LIN {X 0,Y 125.306,Z 694.835,A -85,B 0,C 180,E1 -25457.036,E2 -25457.036} C_VEL
LIN {X 0,Y 123.812,Z 697.112,A -85,B 0,C 180,E1 -25463.481,E2 -25463.481} C_VEL
LIN {X 0,Y 123.139,Z 697.936,A -85,B 0,C 180,E1 -25470,E2 -25470} C_VEL
LIN {X 0,Y 123.809,Z 697.16,A -85,B 0,C 180,E1 -25476.519,E2 -25476.519} C_VEL
LIN {X 0,Y 125.288,Z 694.933,A -85,B 0,C 180,E1 -25482.966,E2 -25482.966} C_VEL
LIN {X 0,Y 127.632,Z 692.097,A -85,B 0,C 180,E1 -25487.629,E2 -25487.629} C_VEL
LIN {X 0,Y 130.588,Z 688.261,A -85,B 0,C 180,E1 -25492.13,E2 -25492.13} C_VEL
LIN {X 0,Y 134.038,Z 683.171,A -85,B 0,C 180,E1 -25496.633,E2 -25496.633} C_VEL
LIN {X 0,Y 137.979,Z 677.127,A -85,B 0,C 180,E1 -25500.62,E2 -25500.62} C_VEL
LIN {X 0,Y 142.589,Z 669.335,A -85,B 0,C 180,E1 -25504.528,E2 -25504.528} C_VEL
LIN {X 0,Y 147.556,Z 659.65,A -85,B 0,C 180,E1 -25508.255,E2 -25508.255} C_VEL
LIN {X 0,Y 151.618,Z 650.591,A -85,B 0,C 180,E1 -25510.899,E2 -25510.899} C_VEL
LIN {X 0,Y 156.205,Z 639.02,A -85,B 0,C 180,E1 -25513.402,E2 -25513.402} C_VEL
LIN {X 0,Y 159.797,Z 627.372,A -85,B 0,C 180,E1 -25515.368,E2 -25515.368} C_VEL
LIN {X 0,Y 162.681,Z 615.545,A -85,B 0,C 180,E1 -25516.802,E2 -25516.802} C_VEL
LIN {X 0,Y 164.589,Z 602.681,A -85,B 0,C 180,E1 -25518.039,E2 -25518.039} C_VEL
LIN {X 0,Y 165.697,Z 590.213,A -85,B 0,C 180,E1 -25518.804,E2 -25518.804} C_VEL
LIN {X 0,Y 166.609,Z 571.79,A -85,B 0,C 180,E1 -25519.65,E2 -25519.65} C_VEL
LIN {X 0,Y 161.362,Z 561.441,A -85,B 0,C 180,E1 -25522.733,E2 -25522.733} C_VEL
LIN {X 0,Y 156.028,Z 552.146,A -85,B 0,C 180,E1 -25526.256,E2 -25526.256} C_VEL
LIN {X 0,Y 151.661,Z 545.284,A -85,B 0,C 180,E1 -25529.556,E2 -25529.556} C_VEL
LIN {X 0,Y 148.447,Z 540.617,A -85,B 0,C 180,E1 -25532.318,E2 -25532.318} C_VEL
LIN {X 0,Y 145.829,Z 537.015,A -85,B 0,C 180,E1 -25534.861,E2 -25534.861} C_VEL
LIN {X 0,Y 143.17,Z 533.482,A -85,B 0,C 180,E1 -25537.829,E2 -25537.829} C_VEL
LIN {X 0,Y 142.512,Z 532.415,A -85,B 0,C 180,E1 -25538.672,E2 -25538.672} C_VEL
LIN {X 0,Y 140.116,Z 529.937,A -85,B 0,C 180,E1 -25541.919,E2 -25541.919} C_VEL
LIN {X 0,Y 138.65,Z 527.238,A -85,B 0,C 180,E1 -25544.549,E2 -25544.549} C_VEL
LIN {X 0,Y 135.862,Z 524.714,A -85,B 0,C 180,E1 -25551.072,E2 -25551.072} C_VEL
LIN {X 0,Y 134.903,Z 522.132,A -85,B 0,C 180,E1 -25557.761,E2 -25557.761} C_VEL
LIN {X 0,Y 134.928,Z 521.81,A -85,B 0,C 180,E1 -25560,E2 -25560} C_VEL
LIN {X 0,Y 135.097,Z 522.892,A -85,B 0,C 180,E1 -25562.982,E2 -25562.982} C_VEL
LIN {X 0,Y 138.648,Z 527.444,A -85,B 0,C 180,E1 -25573.558,E2 -25573.558} C_VEL
LIN {X 0,Y 140.387,Z 530.729,A -85,B 0,C 180,E1 -25576.636,E2 -25576.636} C_VEL
LIN {X 0,Y 144.122,Z 537.229,A -85,B 0,C 180,E1 -25581.674,E2 -25581.674} C_VEL
LIN {X 0,Y 147.623,Z 543.935,A -85,B 0,C 180,E1 -25585.465,E2 -25585.465} C_VEL
LIN {X 0,Y 150.822,Z 550.425,A -85,B 0,C 180,E1 -25588.436,E2 -25588.436} C_VEL
LIN {X 0,Y 153.946,Z 557.142,A -85,B 0,C 180,E1 -25591.021,E2 -25591.021} C_VEL
LIN {X 0,Y 158.018,Z 566.743,A -85,B 0,C 180,E1 -25594.064,E2 -25594.064} C_VEL
LIN {X 0,Y 161.409,Z 576.189,A -85,B 0,C 180,E1 -25596.43,E2 -25596.43} C_VEL
LIN {X 0,Y 162.087,Z 578.257,A -85,B 0,C 180,E1 -25596.888,E2 -25596.888} C_VEL
LIN {X 0,Y 162.907,Z 608.203,A -85,B 0,C 180,E1 -25599.302,E2 -25599.302} C_VEL
LIN {X 0,Y 162.981,Z 619.724,A -85,B 0,C 180,E1 -25600.096,E2 -25600.096} C_VEL
LIN {X 0,Y 161.369,Z 633.381,A -85,B 0,C 180,E1 -25600.774,E2 -25600.774} C_VEL
LIN {X 0,Y 158.919,Z 645.815,A -85,B 0,C 180,E1 -25601.733,E2 -25601.733} C_VEL
LIN {X 0,Y 156.037,Z 656.834,A -85,B 0,C 180,E1 -25602.955,E2 -25602.955} C_VEL
LIN {X 0,Y 151.954,Z 668.683,A -85,B 0,C 180,E1 -25604.677,E2 -25604.677} C_VEL
LIN {X 0,Y 146.967,Z 680.536,A -85,B 0,C 180,E1 -25607.045,E2 -25607.045} C_VEL
LIN {X 0,Y 142.734,Z 689.116,A -85,B 0,C 180,E1 -25609.278,E2 -25609.278} C_VEL
LIN {X 0,Y 137.87,Z 698.049,A -85,B 0,C 180,E1 -25612.288,E2 -25612.288} C_VEL
LIN {X 0,Y 132.801,Z 706.821,A -85,B 0,C 180,E1 -25616.244,E2 -25616.244} C_VEL
LIN {X 0,Y 128.555,Z 713.893,A -85,B 0,C 180,E1 -25620.527,E2 -25620.527} C_VEL
LIN {X 0,Y 125.022,Z 719.59,A -85,B 0,C 180,E1 -25625.065,E2 -25625.065} C_VEL
LIN {X 0,Y 122.616,Z 724.144,A -85,B 0,C 180,E1 -25629.886,E2 -25629.886} C_VEL
LIN {X 0,Y 121.177,Z 727.643,A -85,B 0,C 180,E1 -25634.872,E2 -25634.872} C_VEL
LIN {X 0,Y 120.787,Z 730.791,A -85,B 0,C 180,E1 -25641.55,E2 -25641.55} C_VEL
LIN {X 0,Y 121.419,Z 732.086,A -85,B 0,C 180,E1 -25646.682,E2 -25646.682} C_VEL
LIN {X 0,Y 122.117,Z 732.42,A -85,B 0,C 180,E1 -25650,E2 -25650} C_VEL
LIN {X 0,Y 121.429,Z 732.072,A -85,B 0,C 180,E1 -25653.318,E2 -25653.318} C_VEL
LIN {X 0,Y 120.759,Z 730.143,A -85,B 0,C 180,E1 -25660.055,E2 -25660.055} C_VEL
LIN {X 0,Y 121.18,Z 727.586,A -85,B 0,C 180,E1 -25665.128,E2 -25665.128} C_VEL
LIN {X 0,Y 122.647,Z 724.065,A -85,B 0,C 180,E1 -25670.109,E2 -25670.109} C_VEL
LIN {X 0,Y 125.085,Z 719.488,A -85,B 0,C 180,E1 -25674.922,E2 -25674.922} C_VEL
LIN {X 0,Y 128.554,Z 713.754,A -85,B 0,C 180,E1 -25679.473,E2 -25679.473} C_VEL
LIN {X 0,Y 132.799,Z 706.649,A -85,B 0,C 180,E1 -25683.757,E2 -25683.757} C_VEL
LIN {X 0,Y 135.921,Z 701.383,A -85,B 0,C 180,E1 -25686.236,E2 -25686.236} C_VEL
LIN {X 0,Y 137.564,Z 697.485,A -85,B 0,C 180,E1 -25687.963,E2 -25687.963} C_VEL
LIN {X 0,Y 138.814,Z 690.741,A -85,B 0,C 180,E1 -25690.95,E2 -25690.95} C_VEL
LIN {X 0,Y 140.224,Z 683.56,A -85,B 0,C 180,E1 -25693.685,E2 -25693.685} C_VEL
LIN {X 0,Y 142.028,Z 678.907,A -85,B 0,C 180,E1 -25694.966,E2 -25694.966} C_VEL
LIN {X 0,Y 147.013,Z 667.262,A -85,B 0,C 180,E1 -25697.306,E2 -25697.306} C_VEL
LIN {X 0,Y 151.212,Z 655.339,A -85,B 0,C 180,E1 -25699.023,E2 -25699.023} C_VEL
LIN {X 0,Y 154.607,Z 642.61,A -85,B 0,C 180,E1 -25700.371,E2 -25700.371} C_VEL
LIN {X 0,Y 157.066,Z 629.589,A -85,B 0,C 180,E1 -25701.309,E2 -25701.309} C_VEL
LIN {X 0,Y 158.216,Z 618.69,A -85,B 0,C 180,E1 -25701.849,E2 -25701.849} C_VEL
LIN {X 0,Y 157.786,Z 586.961,A -85,B 0,C 180,E1 -25704.348,E2 -25704.348} C_VEL
LIN {X 0,Y 157.453,Z 580.228,A -85,B 0,C 180,E1 -25705.02,E2 -25705.02} C_VEL
LIN {X 0,Y 153.782,Z 569.769,A -85,B 0,C 180,E1 -25707.812,E2 -25707.812} C_VEL
LIN {X 0,Y 150.559,Z 561.823,A -85,B 0,C 180,E1 -25710.459,E2 -25710.459} C_VEL
LIN {X 0,Y 147.233,Z 554.175,A -85,B 0,C 180,E1 -25713.509,E2 -25713.509} C_VEL
LIN {X 0,Y 144.191,Z 547.823,A -85,B 0,C 180,E1 -25716.671,E2 -25716.671} C_VEL
LIN {X 0,Y 141.243,Z 541.932,A -85,B 0,C 180,E1 -25720.28,E2 -25720.28} C_VEL
LIN {X 0,Y 137.569,Z 534.878,A -85,B 0,C 180,E1 -25726.144,E2 -25726.144} C_VEL
LIN {X 0,Y 136.741,Z 533.764,A -85,B 0,C 180,E1 -25727.76,E2 -25727.76} C_VEL
LIN {X 0,Y 133.829,Z 528.876,A -85,B 0,C 180,E1 -25738.496,E2 -25738.496} C_VEL
LIN {X 0,Y 133.756,Z 528.586,A -85,B 0,C 180,E1 -25740,E2 -25740} C_VEL
LIN {X 0,Y 133.924,Z 529.552,A -85,B 0,C 180,E1 -25744.892,E2 -25744.892} C_VEL
LIN {X 0,Y 136.671,Z 533.761,A -85,B 0,C 180,E1 -25754.138,E2 -25754.138} C_VEL
LIN {X 0,Y 137.444,Z 534.332,A -85,B 0,C 180,E1 -25755.572,E2 -25755.572} C_VEL
LIN {X 0,Y 139.633,Z 537.994,A -85,B 0,C 180,E1 -25759.301,E2 -25759.301} C_VEL
LIN {X 0,Y 141.113,Z 539.535,A -85,B 0,C 180,E1 -25761.262,E2 -25761.262} C_VEL
LIN {X 0,Y 143.561,Z 543.129,A -85,B 0,C 180,E1 -25764.214,E2 -25764.214} C_VEL
LIN {X 0,Y 144.875,Z 544.981,A -85,B 0,C 180,E1 -25765.615,E2 -25765.615} C_VEL
LIN {X 0,Y 147.5,Z 548.879,A -85,B 0,C 180,E1 -25768.165,E2 -25768.165} C_VEL
LIN {X 0,Y 151.608,Z 555.279,A -85,B 0,C 180,E1 -25771.64,E2 -25771.64} C_VEL
LIN {X 0,Y 156.801,Z 564.449,A -85,B 0,C 180,E1 -25775.442,E2 -25775.442} C_VEL
LIN {X 0,Y 160.843,Z 572.43,A -85,B 0,C 180,E1 -25778.073,E2 -25778.073} C_VEL
LIN {X 0,Y 161.898,Z 574.617,A -85,B 0,C 180,E1 -25778.72,E2 -25778.72} C_VEL
LIN {X 0,Y 160.405,Z 598.06,A -85,B 0,C 180,E1 -25779.851,E2 -25779.851} C_VEL
LIN {X 0,Y 158.623,Z 611.11,A -85,B 0,C 180,E1 -25780.869,E2 -25780.869} C_VEL
LIN {X 0,Y 156.036,Z 623.487,A -85,B 0,C 180,E1 -25782.265,E2 -25782.265} C_VEL
LIN {X 0,Y 152.82,Z 634.629,A -85,B 0,C 180,E1 -25783.94,E2 -25783.94} C_VEL
LIN {X 0,Y 148.976,Z 644.988,A -85,B 0,C 180,E1 -25785.907,E2 -25785.907} C_VEL
LIN {X 0,Y 144.507,Z 655.294,A -85,B 0,C 180,E1 -25788.5,E2 -25788.5} C_VEL
LIN {X 0,Y 140.323,Z 663.695,A -85,B 0,C 180,E1 -25791.241,E2 -25791.241} C_VEL
LIN {X 0,Y 136.036,Z 671.414,A -85,B 0,C 180,E1 -25794.465,E2 -25794.465} C_VEL
LIN {X 0,Y 131.173,Z 679.072,A -85,B 0,C 180,E1 -25798.598,E2 -25798.598} C_VEL
LIN {X 0,Y 126.465,Z 685.867,A -85,B 0,C 180,E1 -25803.604,E2 -25803.604} C_VEL
LIN {X 0,Y 122.952,Z 690.47,A -85,B 0,C 180,E1 -25808.19,E2 -25808.19} C_VEL
LIN {X 0,Y 119.998,Z 694.005,A -85,B 0,C 180,E1 -25812.972,E2 -25812.972} C_VEL
LIN {X 0,Y 118.466,Z 695.825,A -85,B 0,C 180,E1 -25816.273,E2 -25816.273} C_VEL
LIN {X 0,Y 116.832,Z 698.101,A -85,B 0,C 180,E1 -25823.09,E2 -25823.09} C_VEL
LIN {X 0,Y 116.111,Z 698.924,A -85,B 0,C 180,E1 -25830,E2 -25830} C_VEL
LIN {X 0,Y 116.829,Z 698.147,A -85,B 0,C 180,E1 -25836.91,E2 -25836.91} C_VEL
LIN {X 0,Y 118.447,Z 695.921,A -85,B 0,C 180,E1 -25843.729,E2 -25843.729} C_VEL
LIN {X 0,Y 120.953,Z 693.084,A -85,B 0,C 180,E1 -25848.637,E2 -25848.637} C_VEL
LIN {X 0,Y 124.106,Z 689.248,A -85,B 0,C 180,E1 -25853.353,E2 -25853.353} C_VEL
LIN {X 0,Y 127.794,Z 684.157,A -85,B 0,C 180,E1 -25858.046,E2 -25858.046} C_VEL
LIN {X 0,Y 131.979,Z 678.113,A -85,B 0,C 180,E1 -25862.174,E2 -25862.174} C_VEL
LIN {X 0,Y 136.857,Z 670.321,A -85,B 0,C 180,E1 -25866.196,E2 -25866.196} C_VEL
LIN {X 0,Y 142.102,Z 660.635,A -85,B 0,C 180,E1 -25870.011,E2 -25870.011} C_VEL
LIN {X 0,Y 146.391,Z 651.573,A -85,B 0,C 180,E1 -25872.696,E2 -25872.696} C_VEL
LIN {X 0,Y 151.168,Z 640.005,A -85,B 0,C 180,E1 -25875.235,E2 -25875.235} C_VEL
LIN {X 0,Y 154.94,Z 628.354,A -85,B 0,C 180,E1 -25877.217,E2 -25877.217} C_VEL
LIN {X 0,Y 157.956,Z 616.524,A -85,B 0,C 180,E1 -25878.66,E2 -25878.66} C_VEL
LIN {X 0,Y 159.983,Z 603.655,A -85,B 0,C 180,E1 -25879.907,E2 -25879.907} C_VEL
LIN {X 0,Y 161.14,Z 591.317,A -85,B 0,C 180,E1 -25880.68,E2 -25880.68} C_VEL
LIN {X 0,Y 162.007,Z 574.666,A -85,B 0,C 180,E1 -25881.471,E2 -25881.471} C_VEL
LIN {X 0,Y 157.105,Z 564.84,A -85,B 0,C 180,E1 -25884.632,E2 -25884.632} C_VEL
LIN {X 0,Y 152.05,Z 555.91,A -85,B 0,C 180,E1 -25888.321,E2 -25888.321} C_VEL
LIN {X 0,Y 148.264,Z 549.964,A -85,B 0,C 180,E1 -25891.485,E2 -25891.485} C_VEL
LIN {X 0,Y 146.224,Z 546.783,A -85,B 0,C 180,E1 -25893.411,E2 -25893.411} C_VEL
LIN {X 0,Y 143.926,Z 543.456,A -85,B 0,C 180,E1 -25895.798,E2 -25895.798} C_VEL
LIN {X 0,Y 141.295,Z 539.731,A -85,B 0,C 180,E1 -25898.957,E2 -25898.957} C_VEL
LIN {X 0,Y 140.514,Z 538.795,A -85,B 0,C 180,E1 -25899.991,E2 -25899.991} C_VEL
LIN {X 0,Y 138.102,Z 535.606,A -85,B 0,C 180,E1 -25903.746,E2 -25903.746} C_VEL
LIN {X 0,Y 137.4,Z 534.069,A -85,B 0,C 180,E1 -25905.182,E2 -25905.182} C_VEL
LIN {X 0,Y 134.994,Z 531.871,A -85,B 0,C 180,E1 -25911.014,E2 -25911.014} C_VEL
LIN {X 0,Y 134.034,Z 529.214,A -85,B 0,C 180,E1 -25917.746,E2 -25917.746} C_VEL
LIN {X 0,Y 134.059,Z 528.886,A -85,B 0,C 180,E1 -25920,E2 -25920} C_VEL
LIN {X 0,Y 134.32,Z 530.461,A -85,B 0,C 180,E1 -25923.844,E2 -25923.844} C_VEL
LIN {X 0,Y 137.485,Z 534.456,A -85,B 0,C 180,E1 -25933.111,E2 -25933.111} C_VEL
LIN {X 0,Y 138.799,Z 537.246,A -85,B 0,C 180,E1 -25935.634,E2 -25935.634} C_VEL
LIN {X 0,Y 142.012,Z 543.19,A -85,B 0,C 180,E1 -25940.364,E2 -25940.364} C_VEL
LIN {X 0,Y 145.325,Z 549.957,A -85,B 0,C 180,E1 -25944.272,E2 -25944.272} C_VEL
LIN {X 0,Y 148.193,Z 556.138,A -85,B 0,C 180,E1 -25947.159,E2 -25947.159} C_VEL
LIN {X 0,Y 150.951,Z 562.491,A -85,B 0,C 180,E1 -25949.645,E2 -25949.645} C_VEL
LIN {X 0,Y 154.757,Z 571.953,A -85,B 0,C 180,E1 -25952.732,E2 -25952.732} C_VEL
LIN {X 0,Y 157.739,Z 580.851,A -85,B 0,C 180,E1 -25955.005,E2 -25955.005} C_VEL
LIN {X 0,Y 158.239,Z 601.084,A -85,B 0,C 180,E1 -25956.749,E2 -25956.749} C_VEL
LIN {X 0,Y 158.364,Z 620.093,A -85,B 0,C 180,E1 -25958.181,E2 -25958.181} C_VEL
LIN {X 0,Y 156.581,Z 633.798,A -85,B 0,C 180,E1 -25958.895,E2 -25958.895} C_VEL
LIN {X 0,Y 154.056,Z 645.721,A -85,B 0,C 180,E1 -25959.839,E2 -25959.839} C_VEL
LIN {X 0,Y 150.662,Z 657.743,A -85,B 0,C 180,E1 -25961.221,E2 -25961.221} C_VEL
LIN {X 0,Y 146.448,Z 669.123,A -85,B 0,C 180,E1 -25962.96,E2 -25962.96} C_VEL
LIN {X 0,Y 141.861,Z 679.544,A -85,B 0,C 180,E1 -25965.094,E2 -25965.094} C_VEL
LIN {X 0,Y 136.354,Z 690.082,A -85,B 0,C 180,E1 -25967.93,E2 -25967.93} C_VEL
LIN {X 0,Y 131.356,Z 698.656,A -85,B 0,C 180,E1 -25971.049,E2 -25971.049} C_VEL
LIN {X 0,Y 126.103,Z 707.082,A -85,B 0,C 180,E1 -25975.163,E2 -25975.163} C_VEL
LIN {X 0,Y 121.199,Z 714.774,A -85,B 0,C 180,E1 -25980.286,E2 -25980.286} C_VEL
LIN {X 0,Y 117.528,Z 720.24,A -85,B 0,C 180,E1 -25985.255,E2 -25985.255} C_VEL
LIN {X 0,Y 115.239,Z 724.436,A -85,B 0,C 180,E1 -25990.402,E2 -25990.402} C_VEL
LIN {X 0,Y 113.977,Z 727.609,A -85,B 0,C 180,E1 -25995.721,E2 -25995.721} C_VEL
LIN {X 0,Y 113.813,Z 730.324,A -85,B 0,C 180,E1 -26002.906,E2 -26002.906} C_VEL
LIN {X 0,Y 114.312,Z 731.086,A -85,B 0,C 180,E1 -26006.475,E2 -26006.475} C_VEL
LIN {X 0,Y 115.024,Z 731.423,A -85,B 0,C 180,E1 -26010,E2 -26010} C_VEL
LIN {X 0,Y 114.322,Z 731.071,A -85,B 0,C 180,E1 -26013.524,E2 -26013.524} C_VEL
LIN {X 0,Y 113.706,Z 729.134,A -85,B 0,C 180,E1 -26020.686,E2 -26020.686} C_VEL
LIN {X 0,Y 114.274,Z 726.577,A -85,B 0,C 180,E1 -26026.066,E2 -26026.066} C_VEL
LIN {X 0,Y 115.948,Z 723.057,A -85,B 0,C 180,E1 -26031.326,E2 -26031.326} C_VEL
LIN {X 0,Y 118.648,Z 718.483,A -85,B 0,C 180,E1 -26036.375,E2 -26036.375} C_VEL
LIN {X 0,Y 123.081,Z 711.682,A -85,B 0,C 180,E1 -26041.882,E2 -26041.882} C_VEL
LIN {X 0,Y 127.775,Z 704.281,A -85,B 0,C 180,E1 -26046.247,E2 -26046.247} C_VEL
LIN {X 0,Y 133.308,Z 695.168,A -85,B 0,C 180,E1 -26050.226,E2 -26050.226} C_VEL
LIN {X 0,Y 138.569,Z 685.87,A -85,B 0,C 180,E1 -26053.211,E2 -26053.211} C_VEL
LIN {X 0,Y 142.028,Z 678.907,A -85,B 0,C 180,E1 -26054.966,E2 -26054.966} C_VEL
LIN {X 0,Y 143.784,Z 674.125,A -85,B 0,C 180,E1 -26056.158,E2 -26056.158} C_VEL
LIN {X 0,Y 145.037,Z 666.088,A -85,B 0,C 180,E1 -26058.404,E2 -26058.404} C_VEL
LIN {X 0,Y 146.023,Z 657.753,A -85,B 0,C 180,E1 -26060.469,E2 -26060.469} C_VEL
LIN {X 0,Y 147.288,Z 652.379,A -85,B 0,C 180,E1 -26061.346,E2 -26061.346} C_VEL
LIN {X 0,Y 150.445,Z 640.418,A -85,B 0,C 180,E1 -26062.573,E2 -26062.573} C_VEL
LIN {X 0,Y 152.757,Z 628.241,A -85,B 0,C 180,E1 -26063.414,E2 -26063.414} C_VEL
LIN {X 0,Y 153.746,Z 619.771,A -85,B 0,C 180,E1 -26063.833,E2 -26063.833} C_VEL
LIN {X 0,Y 153.615,Z 588.769,A -85,B 0,C 180,E1 -26066.347,E2 -26066.347} C_VEL
LIN {X 0,Y 153.37,Z 583.168,A -85,B 0,C 180,E1 -26066.935,E2 -26066.935} C_VEL
LIN {X 0,Y 149.942,Z 572.904,A -85,B 0,C 180,E1 -26069.841,E2 -26069.841} C_VEL
LIN {X 0,Y 146.176,Z 563.414,A -85,B 0,C 180,E1 -26073.342,E2 -26073.342} C_VEL
LIN {X 0,Y 143.565,Z 557.46,A -85,B 0,C 180,E1 -26076.084,E2 -26076.084} C_VEL
LIN {X 0,Y 141.798,Z 553.442,A -85,B 0,C 180,E1 -26078.176,E2 -26078.176} C_VEL
LIN {X 0,Y 139.262,Z 547.958,A -85,B 0,C 180,E1 -26081.614,E2 -26081.614} C_VEL
LIN {X 0,Y 136.049,Z 541.244,A -85,B 0,C 180,E1 -26087.318,E2 -26087.318} C_VEL
LIN {X 0,Y 132.915,Z 535.783,A -85,B 0,C 180,E1 -26099.243,E2 -26099.243} C_VEL
LIN {X 0,Y 132.898,Z 536.075,A -85,B 0,C 180,E1 -26103.032,E2 -26103.032} C_VEL
LIN {X 0,Y 133.914,Z 538.914,A -85,B 0,C 180,E1 -26109.441,E2 -26109.441} C_VEL
LIN {X 0,Y 136.184,Z 541.318,A -85,B 0,C 180,E1 -26114.954,E2 -26114.954} C_VEL
LIN {X 0,Y 138.357,Z 544.887,A -85,B 0,C 180,E1 -26118.812,E2 -26118.812} C_VEL
LIN {X 0,Y 139.518,Z 546.276,A -85,B 0,C 180,E1 -26120.453,E2 -26120.453} C_VEL
LIN {X 0,Y 142.68,Z 551.006,A -85,B 0,C 180,E1 -26124.374,E2 -26124.374} C_VEL
LIN {X 0,Y 145.587,Z 555.556,A -85,B 0,C 180,E1 -26127.394,E2 -26127.394} C_VEL
LIN {X 0,Y 149.369,Z 561.841,A -85,B 0,C 180,E1 -26130.785,E2 -26130.785} C_VEL
LIN {X 0,Y 153.793,Z 570.021,A -85,B 0,C 180,E1 -26134.24,E2 -26134.24} C_VEL
LIN {X 0,Y 157.435,Z 577.581,A -85,B 0,C 180,E1 -26136.794,E2 -26136.794} C_VEL
LIN {X 0,Y 155.973,Z 599.313,A -85,B 0,C 180,E1 -26137.888,E2 -26137.888} C_VEL
LIN {X 0,Y 154.065,Z 612.335,A -85,B 0,C 180,E1 -26138.908,E2 -26138.908} C_VEL
LIN {X 0,Y 151.398,Z 624.482,A -85,B 0,C 180,E1 -26140.296,E2 -26140.296} C_VEL
LIN {X 0,Y 148.03,Z 635.623,A -85,B 0,C 180,E1 -26141.981,E2 -26141.981} C_VEL
LIN {X 0,Y 144.01,Z 645.98,A -85,B 0,C 180,E1 -26143.961,E2 -26143.961} C_VEL
LIN {X 0,Y 139.32,Z 656.286,A -85,B 0,C 180,E1 -26146.584,E2 -26146.584} C_VEL
LIN {X 0,Y 134.914,Z 664.687,A -85,B 0,C 180,E1 -26149.372,E2 -26149.372} C_VEL
LIN {X 0,Y 130.38,Z 672.405,A -85,B 0,C 180,E1 -26152.67,E2 -26152.67} C_VEL
LIN {X 0,Y 125.228,Z 680.062,A -85,B 0,C 180,E1 -26156.923,E2 -26156.923} C_VEL
LIN {X 0,Y 120.21,Z 686.857,A -85,B 0,C 180,E1 -26162.115,E2 -26162.115} C_VEL
LIN {X 0,Y 116.457,Z 691.459,A -85,B 0,C 180,E1 -26166.905,E2 -26166.905} C_VEL
LIN {X 0,Y 113.295,Z 694.994,A -85,B 0,C 180,E1 -26171.931,E2 -26171.931} C_VEL
LIN {X 0,Y 111.649,Z 696.814,A -85,B 0,C 180,E1 -26175.417,E2 -26175.417} C_VEL
LIN {X 0,Y 109.858,Z 699.089,A -85,B 0,C 180,E1 -26182.649,E2 -26182.649} C_VEL
LIN {X 0,Y 109.083,Z 699.913,A -85,B 0,C 180,E1 -26190,E2 -26190} C_VEL
LIN {X 0,Y 109.855,Z 699.135,A -85,B 0,C 180,E1 -26197.351,E2 -26197.351} C_VEL
LIN {X 0,Y 111.63,Z 696.908,A -85,B 0,C 180,E1 -26204.586,E2 -26204.586} C_VEL
LIN {X 0,Y 114.316,Z 694.071,A -85,B 0,C 180,E1 -26209.763,E2 -26209.763} C_VEL
LIN {X 0,Y 117.687,Z 690.235,A -85,B 0,C 180,E1 -26214.709,E2 -26214.709} C_VEL
LIN {X 0,Y 121.636,Z 685.144,A -85,B 0,C 180,E1 -26219.602,E2 -26219.602} C_VEL
LIN {X 0,Y 126.086,Z 679.1,A -85,B 0,C 180,E1 -26223.875,E2 -26223.875} C_VEL
LIN {X 0,Y 131.251,Z 671.307,A -85,B 0,C 180,E1 -26228.008,E2 -26228.008} C_VEL
LIN {X 0,Y 136.793,Z 661.621,A -85,B 0,C 180,E1 -26231.904,E2 -26231.904} C_VEL
LIN {X 0,Y 141.312,Z 652.556,A -85,B 0,C 180,E1 -26234.626,E2 -26234.626} C_VEL
LIN {X 0,Y 146.31,Z 640.989,A -85,B 0,C 180,E1 -26237.186,E2 -26237.186} C_VEL
LIN {X 0,Y 150.255,Z 629.336,A -85,B 0,C 180,E1 -26239.185,E2 -26239.185} C_VEL
LIN {X 0,Y 153.405,Z 617.503,A -85,B 0,C 180,E1 -26240.631,E2 -26240.631} C_VEL
LIN {X 0,Y 155.54,Z 604.644,A -85,B 0,C 180,E1 -26241.891,E2 -26241.891} C_VEL
LIN {X 0,Y 156.781,Z 592.285,A -85,B 0,C 180,E1 -26242.667,E2 -26242.667} C_VEL
LIN {X 0,Y 157.52,Z 577.558,A -85,B 0,C 180,E1 -26243.425,E2 -26243.425} C_VEL
LIN {X 0,Y 153.303,Z 568.852,A -85,B 0,C 180,E1 -26246.423,E2 -26246.423} C_VEL
LIN {X 0,Y 148.732,Z 560.486,A -85,B 0,C 180,E1 -26250.096,E2 -26250.096} C_VEL
LIN {X 0,Y 144.23,Z 553.147,A -85,B 0,C 180,E1 -26254.36,E2 -26254.36} C_VEL
LIN {X 0,Y 141.972,Z 549.781,A -85,B 0,C 180,E1 -26256.863,E2 -26256.863} C_VEL
LIN {X 0,Y 139.27,Z 545.693,A -85,B 0,C 180,E1 -26260.41,E2 -26260.41} C_VEL
LIN {X 0,Y 136.831,Z 542.531,A -85,B 0,C 180,E1 -26264.356,E2 -26264.356} C_VEL
LIN {X 0,Y 136.119,Z 540.967,A -85,B 0,C 180,E1 -26265.899,E2 -26265.899} C_VEL
LIN {X 0,Y 133.61,Z 538.025,A -85,B 0,C 180,E1 -26273.203,E2 -26273.203} C_VEL
LIN {X 0,Y 133.157,Z 536.128,A -85,B 0,C 180,E1 -26278.488,E2 -26278.488} C_VEL
LIN {X 0,Y 133.202,Z 536.104,A -85,B 0,C 180,E1 -26280.567,E2 -26280.567} C_VEL
LIN {X 0,Y 136.244,Z 541.333,A -85,B 0,C 180,E1 -26292.475,E2 -26292.475} C_VEL
LIN {X 0,Y 139.885,Z 548.883,A -85,B 0,C 180,E1 -26298.87,E2 -26298.87} C_VEL
LIN {X 0,Y 143.088,Z 555.973,A -85,B 0,C 180,E1 -26303.037,E2 -26303.037} C_VEL
LIN {X 0,Y 145.715,Z 562.073,A -85,B 0,C 180,E1 -26305.919,E2 -26305.919} C_VEL
LIN {X 0,Y 148.77,Z 569.472,A -85,B 0,C 180,E1 -26308.865,E2 -26308.865} C_VEL
LIN {X 0,Y 152.477,Z 579.869,A -85,B 0,C 180,E1 -26312.101,E2 -26312.101} C_VEL
LIN {X 0,Y 153.727,Z 584.322,A -85,B 0,C 180,E1 -26313.174,E2 -26313.174} C_VEL
LIN {X 0,Y 154.001,Z 614.296,A -85,B 0,C 180,E1 -26315.684,E2 -26315.684} C_VEL
LIN {X 0,Y 153.836,Z 621.406,A -85,B 0,C 180,E1 -26316.193,E2 -26316.193} C_VEL
LIN {X 0,Y 151.8,Z 635.044,A -85,B 0,C 180,E1 -26316.954,E2 -26316.954} C_VEL
LIN {X 0,Y 148.603,Z 648.525,A -85,B 0,C 180,E1 -26318.15,E2 -26318.15} C_VEL
LIN {X 0,Y 144.811,Z 660.299,A -85,B 0,C 180,E1 -26319.607,E2 -26319.607} C_VEL
LIN {X 0,Y 140.477,Z 670.99,A -85,B 0,C 180,E1 -26321.373,E2 -26321.373} C_VEL
LIN {X 0,Y 135.735,Z 680.866,A -85,B 0,C 180,E1 -26323.542,E2 -26323.542} C_VEL
LIN {X 0,Y 130.048,Z 690.895,A -85,B 0,C 180,E1 -26326.448,E2 -26326.448} C_VEL
LIN {X 0,Y 124.907,Z 699.17,A -85,B 0,C 180,E1 -26329.681,E2 -26329.681} C_VEL
LIN {X 0,Y 119.466,Z 707.346,A -85,B 0,C 180,E1 -26333.966,E2 -26333.966} C_VEL
LIN {X 0,Y 115.273,Z 713.397,A -85,B 0,C 180,E1 -26338.222,E2 -26338.222} C_VEL
LIN {X 0,Y 111.074,Z 719.236,A -85,B 0,C 180,E1 -26343.711,E2 -26343.711} C_VEL
LIN {X 0,Y 108.517,Z 723.429,A -85,B 0,C 180,E1 -26349.133,E2 -26349.133} C_VEL
LIN {X 0,Y 107.028,Z 726.599,A -85,B 0,C 180,E1 -26354.772,E2 -26354.772} C_VEL
LIN {X 0,Y 106.73,Z 729.32,A -85,B 0,C 180,E1 -26362.433,E2 -26362.433} C_VEL
LIN {X 0,Y 107.191,Z 730.083,A -85,B 0,C 180,E1 -26366.241,E2 -26366.241} C_VEL
LIN {X 0,Y 107.928,Z 730.426,A -85,B 0,C 180,E1 -26370,E2 -26370} C_VEL
LIN {X 0,Y 107.201,Z 730.068,A -85,B 0,C 180,E1 -26373.759,E2 -26373.759} C_VEL
LIN {X 0,Y 106.7,Z 728.965,A -85,B 0,C 180,E1 -26378.882,E2 -26378.882} C_VEL
LIN {X 0,Y 107.414,Z 725.57,A -85,B 0,C 180,E1 -26387.123,E2 -26387.123} C_VEL
LIN {X 0,Y 109.309,Z 722.049,A -85,B 0,C 180,E1 -26392.691,E2 -26392.691} C_VEL
LIN {X 0,Y 112.301,Z 717.479,A -85,B 0,C 180,E1 -26397.992,E2 -26397.992} C_VEL
LIN {X 0,Y 116.323,Z 711.741,A -85,B 0,C 180,E1 -26402.939,E2 -26402.939} C_VEL
LIN {X 0,Y 121.17,Z 704.635,A -85,B 0,C 180,E1 -26407.517,E2 -26407.517} C_VEL
LIN {X 0,Y 126.904,Z 695.814,A -85,B 0,C 180,E1 -26411.648,E2 -26411.648} C_VEL
LIN {X 0,Y 132.325,Z 686.844,A -85,B 0,C 180,E1 -26414.726,E2 -26414.726} C_VEL
LIN {X 0,Y 137.563,Z 677.027,A -85,B 0,C 180,E1 -26417.256,E2 -26417.256} C_VEL
LIN {X 0,Y 142.281,Z 666.256,A -85,B 0,C 180,E1 -26419.414,E2 -26419.414} C_VEL
LIN {X 0,Y 146.545,Z 654.693,A -85,B 0,C 180,E1 -26421.073,E2 -26421.073} C_VEL
LIN {X 0,Y 147.288,Z 652.379,A -85,B 0,C 180,E1 -26421.346,E2 -26421.346} C_VEL
LIN {X 0,Y 148.432,Z 646.963,A -85,B 0,C 180,E1 -26422.149,E2 -26422.149} C_VEL
LIN {X 0,Y 148.777,Z 638.029,A -85,B 0,C 180,E1 -26423.81,E2 -26423.81} C_VEL
LIN {X 0,Y 148.789,Z 628.889,A -85,B 0,C 180,E1 -26425.295,E2 -26425.295} C_VEL
LIN {X 0,Y 149.247,Z 623.151,A -85,B 0,C 180,E1 -26425.802,E2 -26425.802} C_VEL
LIN {X 0,Y 149.614,Z 610.722,A -85,B 0,C 180,E1 -26426.75,E2 -26426.75} C_VEL
LIN {X 0,Y 149.548,Z 586.46,A -85,B 0,C 180,E1 -26428.872,E2 -26428.872} C_VEL
LIN {X 0,Y 146.439,Z 576.726,A -85,B 0,C 180,E1 -26431.808,E2 -26431.808} C_VEL
LIN {X 0,Y 143.225,Z 568.084,A -85,B 0,C 180,E1 -26435.155,E2 -26435.155} C_VEL
LIN {X 0,Y 140.036,Z 560.057,A -85,B 0,C 180,E1 -26439.048,E2 -26439.048} C_VEL
LIN {X 0,Y 137.414,Z 554.096,A -85,B 0,C 180,E1 -26442.898,E2 -26442.898} C_VEL
LIN {X 0,Y 134.704,Z 547.872,A -85,B 0,C 180,E1 -26448.234,E2 -26448.234} C_VEL
LIN {X 0,Y 132.049,Z 542.839,A -85,B 0,C 180,E1 -26459.238,E2 -26459.238} C_VEL
LIN {X 0,Y 132.033,Z 543.132,A -85,B 0,C 180,E1 -26463.051,E2 -26463.051} C_VEL
LIN {X 0,Y 134.612,Z 547.75,A -85,B 0,C 180,E1 -26473.588,E2 -26473.588} C_VEL
LIN {X 0,Y 137.365,Z 552.075,A -85,B 0,C 180,E1 -26478.727,E2 -26478.727} C_VEL
LIN {X 0,Y 140.693,Z 557.245,A -85,B 0,C 180,E1 -26483.262,E2 -26483.262} C_VEL
LIN {X 0,Y 144.028,Z 562.737,A -85,B 0,C 180,E1 -26486.929,E2 -26486.929} C_VEL
LIN {X 0,Y 147.811,Z 569.545,A -85,B 0,C 180,E1 -26490.466,E2 -26490.466} C_VEL
LIN {X 0,Y 152.221,Z 578.406,A -85,B 0,C 180,E1 -26494.043,E2 -26494.043} C_VEL
LIN {X 0,Y 153.211,Z 580.567,A -85,B 0,C 180,E1 -26494.787,E2 -26494.787} C_VEL
LIN {X 0,Y 151.771,Z 600.184,A -85,B 0,C 180,E1 -26495.783,E2 -26495.783} C_VEL
LIN {X 0,Y 149.857,Z 612.81,A -85,B 0,C 180,E1 -26496.772,E2 -26496.772} C_VEL
LIN {X 0,Y 147.242,Z 624.314,A -85,B 0,C 180,E1 -26498.046,E2 -26498.046} C_VEL
LIN {X 0,Y 143.705,Z 635.831,A -85,B 0,C 180,E1 -26499.752,E2 -26499.752} C_VEL
LIN {X 0,Y 139.224,Z 646.972,A -85,B 0,C 180,E1 -26501.879,E2 -26501.879} C_VEL
LIN {X 0,Y 134.301,Z 657.278,A -85,B 0,C 180,E1 -26504.522,E2 -26504.522} C_VEL
LIN {X 0,Y 129.66,Z 665.678,A -85,B 0,C 180,E1 -26507.35,E2 -26507.35} C_VEL
LIN {X 0,Y 124.865,Z 673.395,A -85,B 0,C 180,E1 -26510.714,E2 -26510.714} C_VEL
LIN {X 0,Y 119.401,Z 681.052,A -85,B 0,C 180,E1 -26515.082,E2 -26515.082} C_VEL
LIN {X 0,Y 114.046,Z 687.846,A -85,B 0,C 180,E1 -26520.463,E2 -26520.463} C_VEL
LIN {X 0,Y 110.026,Z 692.449,A -85,B 0,C 180,E1 -26525.469,E2 -26525.469} C_VEL
LIN {X 0,Y 106.634,Z 695.983,A -85,B 0,C 180,E1 -26530.76,E2 -26530.76} C_VEL
LIN {X 0,Y 104.86,Z 697.803,A -85,B 0,C 180,E1 -26534.45,E2 -26534.45} C_VEL
LIN {X 0,Y 102.891,Z 700.078,A -85,B 0,C 180,E1 -26542.148,E2 -26542.148} C_VEL
LIN {X 0,Y 102.055,Z 700.901,A -85,B 0,C 180,E1 -26550,E2 -26550} C_VEL
LIN {X 0,Y 102.888,Z 700.123,A -85,B 0,C 180,E1 -26557.852,E2 -26557.852} C_VEL
LIN {X 0,Y 104.841,Z 697.896,A -85,B 0,C 180,E1 -26565.553,E2 -26565.553} C_VEL
LIN {X 0,Y 107.728,Z 695.058,A -85,B 0,C 180,E1 -26571.027,E2 -26571.027} C_VEL
LIN {X 0,Y 111.341,Z 691.222,A -85,B 0,C 180,E1 -26576.221,E2 -26576.221} C_VEL
LIN {X 0,Y 115.578,Z 686.131,A -85,B 0,C 180,E1 -26581.324,E2 -26581.324} C_VEL
LIN {X 0,Y 120.315,Z 680.086,A -85,B 0,C 180,E1 -26585.741,E2 -26585.741} C_VEL
LIN {X 0,Y 125.787,Z 672.292,A -85,B 0,C 180,E1 -26589.98,E2 -26589.98} C_VEL
LIN {X 0,Y 131.645,Z 662.606,A -85,B 0,C 180,E1 -26593.948,E2 -26593.948} C_VEL
LIN {X 0,Y 136.401,Z 653.54,A -85,B 0,C 180,E1 -26596.699,E2 -26596.699} C_VEL
LIN {X 0,Y 141.629,Z 641.97,A -85,B 0,C 180,E1 -26599.272,E2 -26599.272} C_VEL
LIN {X 0,Y 145.759,Z 630.318,A -85,B 0,C 180,E1 -26601.276,E2 -26601.276} C_VEL
LIN {X 0,Y 149.046,Z 618.483,A -85,B 0,C 180,E1 -26602.72,E2 -26602.72} C_VEL
LIN {X 0,Y 151.294,Z 605.772,A -85,B 0,C 180,E1 -26603.967,E2 -26603.967} C_VEL
LIN {X 0,Y 152.497,Z 594.334,A -85,B 0,C 180,E1 -26604.728,E2 -26604.728} C_VEL
LIN {X 0,Y 153.365,Z 580.698,A -85,B 0,C 180,E1 -26605.393,E2 -26605.393} C_VEL
LIN {X 0,Y 149.009,Z 571.618,A -85,B 0,C 180,E1 -26608.842,E2 -26608.842} C_VEL
LIN {X 0,Y 145.028,Z 564.285,A -85,B 0,C 180,E1 -26612.449,E2 -26612.449} C_VEL
LIN {X 0,Y 141.613,Z 558.527,A -85,B 0,C 180,E1 -26616.082,E2 -26616.082} C_VEL
LIN {X 0,Y 139.837,Z 555.836,A -85,B 0,C 180,E1 -26618.244,E2 -26618.244} C_VEL
LIN {X 0,Y 137.569,Z 552.197,A -85,B 0,C 180,E1 -26621.502,E2 -26621.502} C_VEL
LIN {X 0,Y 135.205,Z 548.638,A -85,B 0,C 180,E1 -26625.801,E2 -26625.801} C_VEL
LIN {X 0,Y 134.835,Z 547.83,A -85,B 0,C 180,E1 -26626.684,E2 -26626.684} C_VEL
LIN {X 0,Y 132.289,Z 543.201,A -85,B 0,C 180,E1 -26638.478,E2 -26638.478} C_VEL
LIN {X 0,Y 132.325,Z 543.154,A -85,B 0,C 180,E1 -26640.38,E2 -26640.38} C_VEL
LIN {X 0,Y 135.02,Z 548.206,A -85,B 0,C 180,E1 -26651.827,E2 -26651.827} C_VEL
LIN {X 0,Y 138.226,Z 555.615,A -85,B 0,C 180,E1 -26657.953,E2 -26657.953} C_VEL
LIN {X 0,Y 140.756,Z 561.6,A -85,B 0,C 180,E1 -26661.552,E2 -26661.552} C_VEL
LIN {X 0,Y 143.387,Z 568.151,A -85,B 0,C 180,E1 -26664.718,E2 -26664.718} C_VEL
LIN {X 0,Y 146.013,Z 575.171,A -85,B 0,C 180,E1 -26667.502,E2 -26667.502} C_VEL
LIN {X 0,Y 149.082,Z 584.37,A -85,B 0,C 180,E1 -26670.449,E2 -26670.449} C_VEL
LIN {X 0,Y 149.809,Z 586.855,A -85,B 0,C 180,E1 -26671.121,E2 -26671.121} C_VEL
LIN {X 0,Y 149.785,Z 617.576,A -85,B 0,C 180,E1 -26673.74,E2 -26673.74} C_VEL
LIN {X 0,Y 149.479,Z 622.759,A -85,B 0,C 180,E1 -26674.093,E2 -26674.093} C_VEL
LIN {X 0,Y 147.152,Z 636.218,A -85,B 0,C 180,E1 -26674.902,E2 -26674.902} C_VEL
LIN {X 0,Y 143.776,Z 649.269,A -85,B 0,C 180,E1 -26676.089,E2 -26676.089} C_VEL
LIN {X 0,Y 139.729,Z 660.981,A -85,B 0,C 180,E1 -26677.612,E2 -26677.612} C_VEL
LIN {X 0,Y 134.619,Z 672.611,A -85,B 0,C 180,E1 -26679.644,E2 -26679.644} C_VEL
LIN {X 0,Y 129.099,Z 683.104,A -85,B 0,C 180,E1 -26682.123,E2 -26682.123} C_VEL
LIN {X 0,Y 123.848,Z 691.701,A -85,B 0,C 180,E1 -26684.821,E2 -26684.821} C_VEL
LIN {X 0,Y 118.547,Z 699.685,A -85,B 0,C 180,E1 -26688.169,E2 -26688.169} C_VEL
LIN {X 0,Y 112.874,Z 707.529,A -85,B 0,C 180,E1 -26692.623,E2 -26692.623} C_VEL
LIN {X 0,Y 107.394,Z 714.835,A -85,B 0,C 180,E1 -26698.432,E2 -26698.432} C_VEL
LIN {X 0,Y 103.631,Z 719.737,A -85,B 0,C 180,E1 -26703.845,E2 -26703.845} C_VEL
LIN {X 0,Y 101.138,Z 723.571,A -85,B 0,C 180,E1 -26709.669,E2 -26709.669} C_VEL
LIN {X 0,Y 100.137,Z 725.593,A -85,B 0,C 180,E1 -26713.696,E2 -26713.696} C_VEL
LIN {X 0,Y 99.673,Z 728.319,A -85,B 0,C 180,E1 -26721.893,E2 -26721.893} C_VEL
LIN {X 0,Y 100.076,Z 729.08,A -85,B 0,C 180,E1 -26725.973,E2 -26725.973} C_VEL
LIN {X 0,Y 100.827,Z 729.427,A -85,B 0,C 180,E1 -26730,E2 -26730} C_VEL
LIN {X 0,Y 100.085,Z 729.065,A -85,B 0,C 180,E1 -26734.027,E2 -26734.027} C_VEL
LIN {X 0,Y 99.636,Z 728.065,A -85,B 0,C 180,E1 -26739.065,E2 -26739.065} C_VEL
LIN {X 0,Y 100.141,Z 725.539,A -85,B 0,C 180,E1 -26746.303,E2 -26746.303} C_VEL
LIN {X 0,Y 101.896,Z 722.352,A -85,B 0,C 180,E1 -26752.293,E2 -26752.293} C_VEL
LIN {X 0,Y 104.773,Z 718.135,A -85,B 0,C 180,E1 -26758.004,E2 -26758.004} C_VEL
LIN {X 0,Y 109.514,Z 711.879,A -85,B 0,C 180,E1 -26764.049,E2 -26764.049} C_VEL
LIN {X 0,Y 114.647,Z 704.892,A -85,B 0,C 180,E1 -26768.927,E2 -26768.927} C_VEL
LIN {X 0,Y 120.603,Z 696.434,A -85,B 0,C 180,E1 -26773.212,E2 -26773.212} C_VEL
LIN {X 0,Y 126.197,Z 687.812,A -85,B 0,C 180,E1 -26776.383,E2 -26776.383} C_VEL
LIN {X 0,Y 131.59,Z 678.387,A -85,B 0,C 180,E1 -26778.971,E2 -26778.971} C_VEL
LIN {X 0,Y 137.124,Z 666.696,A -85,B 0,C 180,E1 -26781.406,E2 -26781.406} C_VEL
LIN {X 0,Y 141.531,Z 655.596,A -85,B 0,C 180,E1 -26783.068,E2 -26783.068} C_VEL
LIN {X 0,Y 145.093,Z 643.975,A -85,B 0,C 180,E1 -26784.376,E2 -26784.376} C_VEL
LIN {X 0,Y 148.062,Z 630.695,A -85,B 0,C 180,E1 -26785.392,E2 -26785.392} C_VEL
LIN {X 0,Y 149.247,Z 623.151,A -85,B 0,C 180,E1 -26785.802,E2 -26785.802} C_VEL
LIN {X 0,Y 149.505,Z 619.337,A -85,B 0,C 180,E1 -26786.114,E2 -26786.114} C_VEL
LIN {X 0,Y 149.279,Z 615.651,A -85,B 0,C 180,E1 -26786.623,E2 -26786.623} C_VEL
LIN {X 0,Y 148.002,Z 608.638,A -85,B 0,C 180,E1 -26787.981,E2 -26787.981} C_VEL
LIN {X 0,Y 146.226,Z 599.844,A -85,B 0,C 180,E1 -26789.778,E2 -26789.778} C_VEL
LIN {X 0,Y 145.836,Z 594.179,A -85,B 0,C 180,E1 -26790.532,E2 -26790.532} C_VEL
LIN {X 0,Y 145.769,Z 589.242,A -85,B 0,C 180,E1 -26791.05,E2 -26791.05} C_VEL
LIN {X 0,Y 142.753,Z 579.343,A -85,B 0,C 180,E1 -26794.287,E2 -26794.287} C_VEL
LIN {X 0,Y 139.738,Z 570.775,A -85,B 0,C 180,E1 -26797.935,E2 -26797.935} C_VEL
LIN {X 0,Y 137.446,Z 564.834,A -85,B 0,C 180,E1 -26801.169,E2 -26801.169} C_VEL
LIN {X 0,Y 135.589,Z 560.107,A -85,B 0,C 180,E1 -26804.306,E2 -26804.306} C_VEL
LIN {X 0,Y 133.445,Z 554.624,A -85,B 0,C 180,E1 -26809.032,E2 -26809.032} C_VEL
LIN {X 0,Y 131.155,Z 549.774,A -85,B 0,C 180,E1 -26820,E2 -26820} C_VEL
LIN {X 0,Y 131.199,Z 550.583,A -85,B 0,C 180,E1 -26823.878,E2 -26823.878} C_VEL
LIN {X 0,Y 133.275,Z 554.501,A -85,B 0,C 180,E1 -26832.611,E2 -26832.611} C_VEL
LIN {X 0,Y 133.8,Z 555.373,A -85,B 0,C 180,E1 -26833.866,E2 -26833.866} C_VEL
LIN {X 0,Y 136.404,Z 559.645,A -85,B 0,C 180,E1 -26838.746,E2 -26838.746} C_VEL
LIN {X 0,Y 138.963,Z 563.88,A -85,B 0,C 180,E1 -26842.389,E2 -26842.389} C_VEL
LIN {X 0,Y 141.451,Z 568.186,A -85,B 0,C 180,E1 -26845.357,E2 -26845.357} C_VEL
LIN {X 0,Y 145.002,Z 574.868,A -85,B 0,C 180,E1 -26848.992,E2 -26848.992} C_VEL
LIN {X 0,Y 149.108,Z 583.57,A -85,B 0,C 180,E1 -26852.623,E2 -26852.623} C_VEL
LIN {X 0,Y 147.597,Z 602.49,A -85,B 0,C 180,E1 -26853.647,E2 -26853.647} C_VEL
LIN {X 0,Y 145.361,Z 615.708,A -85,B 0,C 180,E1 -26854.724,E2 -26854.724} C_VEL
LIN {X 0,Y 142.435,Z 627.357,A -85,B 0,C 180,E1 -26856.106,E2 -26856.106} C_VEL
LIN {X 0,Y 138.586,Z 638.777,A -85,B 0,C 180,E1 -26857.883,E2 -26857.883} C_VEL
LIN {X 0,Y 134.05,Z 649.235,A -85,B 0,C 180,E1 -26859.938,E2 -26859.938} C_VEL
LIN {X 0,Y 129.47,Z 658.27,A -85,B 0,C 180,E1 -26862.304,E2 -26862.304} C_VEL
LIN {X 0,Y 124.582,Z 666.669,A -85,B 0,C 180,E1 -26865.159,E2 -26865.159} C_VEL
LIN {X 0,Y 119.508,Z 674.386,A -85,B 0,C 180,E1 -26868.58,E2 -26868.58} C_VEL
LIN {X 0,Y 113.709,Z 682.042,A -85,B 0,C 180,E1 -26873.054,E2 -26873.054} C_VEL
LIN {X 0,Y 107.987,Z 688.836,A -85,B 0,C 180,E1 -26878.625,E2 -26878.625} C_VEL
LIN {X 0,Y 103.674,Z 693.438,A -85,B 0,C 180,E1 -26883.856,E2 -26883.856} C_VEL
LIN {X 0,Y 100.023,Z 696.972,A -85,B 0,C 180,E1 -26889.433,E2 -26889.433} C_VEL
LIN {X 0,Y 98.105,Z 698.792,A -85,B 0,C 180,E1 -26893.349,E2 -26893.349} C_VEL
LIN {X 0,Y 95.934,Z 701.066,A -85,B 0,C 180,E1 -26901.575,E2 -26901.575} C_VEL
LIN {X 0,Y 95.027,Z 701.889,A -85,B 0,C 180,E1 -26910,E2 -26910} C_VEL
LIN {X 0,Y 95.931,Z 701.111,A -85,B 0,C 180,E1 -26918.425,E2 -26918.425} C_VEL
LIN {X 0,Y 98.086,Z 698.884,A -85,B 0,C 180,E1 -26926.654,E2 -26926.654} C_VEL
LIN {X 0,Y 101.199,Z 696.046,A -85,B 0,C 180,E1 -26932.455,E2 -26932.455} C_VEL
LIN {X 0,Y 105.082,Z 692.209,A -85,B 0,C 180,E1 -26937.915,E2 -26937.915} C_VEL
LIN {X 0,Y 109.635,Z 687.117,A -85,B 0,C 180,E1 -26943.233,E2 -26943.233} C_VEL
LIN {X 0,Y 114.684,Z 681.072,A -85,B 0,C 180,E1 -26947.792,E2 -26947.792} C_VEL
LIN {X 0,Y 120.486,Z 673.278,A -85,B 0,C 180,E1 -26952.127,E2 -26952.127} C_VEL
LIN {X 0,Y 126.678,Z 663.591,A -85,B 0,C 180,E1 -26956.155,E2 -26956.155} C_VEL
LIN {X 0,Y 131.682,Z 654.524,A -85,B 0,C 180,E1 -26958.925,E2 -26958.925} C_VEL
LIN {X 0,Y 137.14,Z 642.956,A -85,B 0,C 180,E1 -26961.502,E2 -26961.502} C_VEL
LIN {X 0,Y 141.468,Z 631.3,A -85,B 0,C 180,E1 -26963.497,E2 -26963.497} C_VEL
LIN {X 0,Y 144.897,Z 619.463,A -85,B 0,C 180,E1 -26964.932,E2 -26964.932} C_VEL
LIN {X 0,Y 147.236,Z 606.958,A -85,B 0,C 180,E1 -26966.162,E2 -26966.162} C_VEL
LIN {X 0,Y 148.539,Z 595.305,A -85,B 0,C 180,E1 -26966.948,E2 -26966.948} C_VEL
LIN {X 0,Y 149.298,Z 583.74,A -85,B 0,C 180,E1 -26967.541,E2 -26967.541} C_VEL
LIN {X 0,Y 145.144,Z 574.871,A -85,B 0,C 180,E1 -26971.237,E2 -26971.237} C_VEL
LIN {X 0,Y 141.295,Z 567.709,A -85,B 0,C 180,E1 -26975.229,E2 -26975.229} C_VEL
LIN {X 0,Y 138.57,Z 562.878,A -85,B 0,C 180,E1 -26978.62,E2 -26978.62} C_VEL
LIN {X 0,Y 135.876,Z 558.614,A -85,B 0,C 180,E1 -26982.698,E2 -26982.698} C_VEL
LIN {X 0,Y 133.589,Z 554.664,A -85,B 0,C 180,E1 -26987.466,E2 -26987.466} C_VEL
LIN {X 0,Y 131.419,Z 550.293,A -85,B 0,C 180,E1 -26998.468,E2 -26998.468} C_VEL
LIN {X 0,Y 131.439,Z 550.334,A -85,B 0,C 180,E1 -27000.287,E2 -27000.287} C_VEL
LIN {X 0,Y 133.741,Z 554.919,A -85,B 0,C 180,E1 -27010.981,E2 -27010.981} C_VEL
LIN {X 0,Y 136.393,Z 561.729,A -85,B 0,C 180,E1 -27016.635,E2 -27016.635} C_VEL
LIN {X 0,Y 138.648,Z 567.556,A -85,B 0,C 180,E1 -27020.201,E2 -27020.201} C_VEL
LIN {X 0,Y 141.481,Z 575.125,A -85,B 0,C 180,E1 -27023.901,E2 -27023.901} C_VEL
LIN {X 0,Y 144.961,Z 585.815,A -85,B 0,C 180,E1 -27027.816,E2 -27027.816} C_VEL
LIN {X 0,Y 146.079,Z 590.137,A -85,B 0,C 180,E1 -27029.024,E2 -27029.024} C_VEL
LIN {X 0,Y 145.723,Z 619.254,A -85,B 0,C 180,E1 -27031.559,E2 -27031.559} C_VEL
LIN {X 0,Y 145.101,Z 625.178,A -85,B 0,C 180,E1 -27031.939,E2 -27031.939} C_VEL
LIN {X 0,Y 142.532,Z 638.183,A -85,B 0,C 180,E1 -27032.789,E2 -27032.789} C_VEL
LIN {X 0,Y 139.26,Z 649.61,A -85,B 0,C 180,E1 -27033.874,E2 -27033.874} C_VEL
LIN {X 0,Y 134.832,Z 661.578,A -85,B 0,C 180,E1 -27035.47,E2 -27035.47} C_VEL
LIN {X 0,Y 129.541,Z 672.916,A -85,B 0,C 180,E1 -27037.493,E2 -27037.493} C_VEL
LIN {X 0,Y 124.45,Z 682.11,A -85,B 0,C 180,E1 -27039.698,E2 -27039.698} C_VEL
LIN {X 0,Y 118.942,Z 690.704,A -85,B 0,C 180,E1 -27042.39,E2 -27042.39} C_VEL
LIN {X 0,Y 113.314,Z 698.681,A -85,B 0,C 180,E1 -27045.755,E2 -27045.755} C_VEL
LIN {X 0,Y 107.283,Z 706.525,A -85,B 0,C 180,E1 -27050.305,E2 -27050.305} C_VEL
LIN {X 0,Y 101.392,Z 713.835,A -85,B 0,C 180,E1 -27056.323,E2 -27056.323} C_VEL
LIN {X 0,Y 97.254,Z 718.731,A -85,B 0,C 180,E1 -27061.985,E2 -27061.985} C_VEL
LIN {X 0,Y 94.444,Z 722.563,A -85,B 0,C 180,E1 -27068.157,E2 -27068.157} C_VEL
LIN {X 0,Y 93.263,Z 724.584,A -85,B 0,C 180,E1 -27072.457,E2 -27072.457} C_VEL
LIN {X 0,Y 92.614,Z 727.316,A -85,B 0,C 180,E1 -27081.271,E2 -27081.271} C_VEL
LIN {X 0,Y 92.97,Z 728.078,A -85,B 0,C 180,E1 -27085.665,E2 -27085.665} C_VEL
LIN {X 0,Y 93.721,Z 728.428,A -85,B 0,C 180,E1 -27090,E2 -27090} C_VEL
LIN {X 0,Y 92.981,Z 728.063,A -85,B 0,C 180,E1 -27094.335,E2 -27094.335} C_VEL
LIN {X 0,Y 92.591,Z 727.154,A -85,B 0,C 180,E1 -27099.338,E2 -27099.338} C_VEL
LIN {X 0,Y 93.269,Z 724.529,A -85,B 0,C 180,E1 -27107.542,E2 -27107.542} C_VEL
LIN {X 0,Y 95.284,Z 721.34,A -85,B 0,C 180,E1 -27113.933,E2 -27113.933} C_VEL
LIN {X 0,Y 98.527,Z 717.13,A -85,B 0,C 180,E1 -27119.954,E2 -27119.954} C_VEL
LIN {X 0,Y 103.756,Z 710.769,A -85,B 0,C 180,E1 -27126.347,E2 -27126.347} C_VEL
LIN {X 0,Y 109.183,Z 703.886,A -85,B 0,C 180,E1 -27131.282,E2 -27131.282} C_VEL
LIN {X 0,Y 115.508,Z 695.429,A -85,B 0,C 180,E1 -27135.635,E2 -27135.635} C_VEL
LIN {X 0,Y 121.381,Z 686.805,A -85,B 0,C 180,E1 -27138.824,E2 -27138.824} C_VEL
LIN {X 0,Y 127.684,Z 676.202,A -85,B 0,C 180,E1 -27141.659,E2 -27141.659} C_VEL
LIN {X 0,Y 132.81,Z 665.693,A -85,B 0,C 180,E1 -27143.802,E2 -27143.802} C_VEL
LIN {X 0,Y 137.706,Z 653.667,A -85,B 0,C 180,E1 -27145.56,E2 -27145.56} C_VEL
LIN {X 0,Y 141.463,Z 641.385,A -85,B 0,C 180,E1 -27146.873,E2 -27146.873} C_VEL
LIN {X 0,Y 144.382,Z 628.195,A -85,B 0,C 180,E1 -27147.832,E2 -27147.832} C_VEL
LIN {X 0,Y 145.428,Z 621.103,A -85,B 0,C 180,E1 -27148.22,E2 -27148.22} C_VEL
LIN {X 0,Y 145.836,Z 594.179,A -85,B 0,C 180,E1 -27150.532,E2 -27150.532} C_VEL
LIN {X 0,Y 145.434,Z 591.389,A -85,B 0,C 180,E1 -27151.071,E2 -27151.071} C_VEL
LIN {X 0,Y 144.48,Z 589.236,A -85,B 0,C 180,E1 -27151.95,E2 -27151.95} C_VEL
LIN {X 0,Y 143.02,Z 587.325,A -85,B 0,C 180,E1 -27153.221,E2 -27153.221} C_VEL
LIN {X 0,Y 139.945,Z 583.684,A -85,B 0,C 180,E1 -27156.146,E2 -27156.146} C_VEL
LIN {X 0,Y 139.219,Z 581.925,A -85,B 0,C 180,E1 -27157.016,E2 -27157.016} C_VEL
LIN {X 0,Y 137.129,Z 575.521,A -85,B 0,C 180,E1 -27159.956,E2 -27159.956} C_VEL
LIN {X 0,Y 135.466,Z 570.707,A -85,B 0,C 180,E1 -27162.644,E2 -27162.644} C_VEL
LIN {X 0,Y 133.889,Z 566.258,A -85,B 0,C 180,E1 -27165.658,E2 -27165.658} C_VEL
LIN {X 0,Y 132.129,Z 561.328,A -85,B 0,C 180,E1 -27170.045,E2 -27170.045} C_VEL
LIN {X 0,Y 130.288,Z 556.83,A -85,B 0,C 180,E1 -27180,E2 -27180} C_VEL
LIN {X 0,Y 130.301,Z 557.559,A -85,B 0,C 180,E1 -27183.498,E2 -27183.498} C_VEL
LIN {X 0,Y 132.098,Z 561.315,A -85,B 0,C 180,E1 -27191.906,E2 -27191.906} C_VEL
LIN {X 0,Y 132.898,Z 562.943,A -85,B 0,C 180,E1 -27193.962,E2 -27193.962} C_VEL
LIN {X 0,Y 134.93,Z 566.348,A -85,B 0,C 180,E1 -27197.917,E2 -27197.917} C_VEL
LIN {X 0,Y 137.268,Z 570.494,A -85,B 0,C 180,E1 -27201.494,E2 -27201.494} C_VEL
LIN {X 0,Y 140.131,Z 575.787,A -85,B 0,C 180,E1 -27205.088,E2 -27205.088} C_VEL
LIN {X 0,Y 143.689,Z 583.255,A -85,B 0,C 180,E1 -27208.882,E2 -27208.882} C_VEL
LIN {X 0,Y 145.273,Z 586.883,A -85,B 0,C 180,E1 -27210.401,E2 -27210.401} C_VEL
LIN {X 0,Y 143.736,Z 604.151,A -85,B 0,C 180,E1 -27211.358,E2 -27211.358} C_VEL
LIN {X 0,Y 141.469,Z 616.706,A -85,B 0,C 180,E1 -27212.38,E2 -27212.38} C_VEL
LIN {X 0,Y 138.409,Z 628.352,A -85,B 0,C 180,E1 -27213.754,E2 -27213.754} C_VEL
LIN {X 0,Y 134.383,Z 639.773,A -85,B 0,C 180,E1 -27215.517,E2 -27215.517} C_VEL
LIN {X 0,Y 129.65,Z 650.228,A -85,B 0,C 180,E1 -27217.556,E2 -27217.556} C_VEL
LIN {X 0,Y 124.847,Z 659.262,A -85,B 0,C 180,E1 -27219.917,E2 -27219.917} C_VEL
LIN {X 0,Y 119.701,Z 667.66,A -85,B 0,C 180,E1 -27222.786,E2 -27222.786} C_VEL
LIN {X 0,Y 114.332,Z 675.376,A -85,B 0,C 180,E1 -27226.249,E2 -27226.249} C_VEL
LIN {X 0,Y 108.175,Z 683.032,A -85,B 0,C 180,E1 -27230.816,E2 -27230.816} C_VEL
LIN {X 0,Y 102.052,Z 689.826,A -85,B 0,C 180,E1 -27236.57,E2 -27236.57} C_VEL
LIN {X 0,Y 97.414,Z 694.427,A -85,B 0,C 180,E1 -27242.035,E2 -27242.035} C_VEL
LIN {X 0,Y 93.474,Z 697.962,A -85,B 0,C 180,E1 -27247.919,E2 -27247.919} C_VEL
LIN {X 0,Y 91.391,Z 699.781,A -85,B 0,C 180,E1 -27252.086,E2 -27252.086} C_VEL
LIN {X 0,Y 88.987,Z 702.055,A -85,B 0,C 180,E1 -27260.912,E2 -27260.912} C_VEL
LIN {X 0,Y 88,Z 702.877,A -85,B 0,C 180,E1 -27270,E2 -27270} C_VEL
LIN {X 0,Y 88.984,Z 702.099,A -85,B 0,C 180,E1 -27279.088,E2 -27279.088} C_VEL
LIN {X 0,Y 91.372,Z 699.872,A -85,B 0,C 180,E1 -27287.918,E2 -27287.918} C_VEL
LIN {X 0,Y 94.742,Z 697.033,A -85,B 0,C 180,E1 -27294.078,E2 -27294.078} C_VEL
LIN {X 0,Y 98.927,Z 693.196,A -85,B 0,C 180,E1 -27299.821,E2 -27299.821} C_VEL
LIN {X 0,Y 103.828,Z 688.104,A -85,B 0,C 180,E1 -27305.359,E2 -27305.359} C_VEL
LIN {X 0,Y 109.215,Z 682.058,A -85,B 0,C 180,E1 -27310.052,E2 -27310.052} C_VEL
LIN {X 0,Y 115.37,Z 674.264,A -85,B 0,C 180,E1 -27314.47,E2 -27314.47} C_VEL
LIN {X 0,Y 121.914,Z 664.577,A -85,B 0,C 180,E1 -27318.538,E2 -27318.538} C_VEL
LIN {X 0,Y 127.175,Z 655.509,A -85,B 0,C 180,E1 -27321.312,E2 -27321.312} C_VEL
LIN {X 0,Y 132.884,Z 643.939,A -85,B 0,C 180,E1 -27323.87,E2 -27323.87} C_VEL
LIN {X 0,Y 137.404,Z 632.282,A -85,B 0,C 180,E1 -27325.854,E2 -27325.854} C_VEL
LIN {X 0,Y 140.966,Z 620.445,A -85,B 0,C 180,E1 -27327.277,E2 -27327.277} C_VEL
LIN {X 0,Y 143.512,Z 607.487,A -85,B 0,C 180,E1 -27328.532,E2 -27328.532} C_VEL
LIN {X 0,Y 144.982,Z 594.613,A -85,B 0,C 180,E1 -27329.362,E2 -27329.362} C_VEL
LIN {X 0,Y 145.47,Z 586.981,A -85,B 0,C 180,E1 -27329.773,E2 -27329.773} C_VEL
LIN {X 0,Y 141.524,Z 578.292,A -85,B 0,C 180,E1 -27333.759,E2 -27333.759} C_VEL
LIN {X 0,Y 137.786,Z 571.091,A -85,B 0,C 180,E1 -27338.297,E2 -27338.297} C_VEL
LIN {X 0,Y 135.858,Z 567.869,A -85,B 0,C 180,E1 -27341.096,E2 -27341.096} C_VEL
LIN {X 0,Y 134.38,Z 565.217,A -85,B 0,C 180,E1 -27343.673,E2 -27343.673} C_VEL
LIN {X 0,Y 132.349,Z 561.46,A -85,B 0,C 180,E1 -27348.319,E2 -27348.319} C_VEL
LIN {X 0,Y 130.548,Z 557.383,A -85,B 0,C 180,E1 -27358.457,E2 -27358.457} C_VEL
LIN {X 0,Y 130.553,Z 557.546,A -85,B 0,C 180,E1 -27360.289,E2 -27360.289} C_VEL
LIN {X 0,Y 132.502,Z 561.726,A -85,B 0,C 180,E1 -27370.167,E2 -27370.167} C_VEL
LIN {X 0,Y 134.659,Z 567.86,A -85,B 0,C 180,E1 -27375.32,E2 -27375.32} C_VEL
LIN {X 0,Y 136.674,Z 573.637,A -85,B 0,C 180,E1 -27378.893,E2 -27378.893} C_VEL
LIN {X 0,Y 139.039,Z 580.684,A -85,B 0,C 180,E1 -27382.353,E2 -27382.353} C_VEL
LIN {X 0,Y 141.908,Z 590.254,A -85,B 0,C 180,E1 -27385.976,E2 -27385.976} C_VEL
LIN {X 0,Y 142.551,Z 593.173,A -85,B 0,C 180,E1 -27386.791,E2 -27386.791} C_VEL
LIN {X 0,Y 141.887,Z 620.751,A -85,B 0,C 180,E1 -27389.255,E2 -27389.255} C_VEL
LIN {X 0,Y 139.941,Z 632.341,A -85,B 0,C 180,E1 -27389.972,E2 -27389.972} C_VEL
LIN {X 0,Y 136.303,Z 645.917,A -85,B 0,C 180,E1 -27391.098,E2 -27391.098} C_VEL
LIN {X 0,Y 132.242,Z 657.319,A -85,B 0,C 180,E1 -27392.472,E2 -27392.472} C_VEL
LIN {X 0,Y 126.698,Z 669.316,A -85,B 0,C 180,E1 -27394.401,E2 -27394.401} C_VEL
LIN {X 0,Y 120.713,Z 680.039,A -85,B 0,C 180,E1 -27396.82,E2 -27396.82} C_VEL
LIN {X 0,Y 114.275,Z 689.708,A -85,B 0,C 180,E1 -27399.759,E2 -27399.759} C_VEL
LIN {X 0,Y 108.315,Z 697.679,A -85,B 0,C 180,E1 -27403.119,E2 -27403.119} C_VEL
LIN {X 0,Y 101.873,Z 705.52,A -85,B 0,C 180,E1 -27407.731,E2 -27407.731} C_VEL
LIN {X 0,Y 95.523,Z 712.831,A -85,B 0,C 180,E1 -27413.944,E2 -27413.944} C_VEL
LIN {X 0,Y 90.991,Z 717.725,A -85,B 0,C 180,E1 -27419.865,E2 -27419.865} C_VEL
LIN {X 0,Y 87.818,Z 721.554,A -85,B 0,C 180,E1 -27426.413,E2 -27426.413} C_VEL
LIN {X 0,Y 86.459,Z 723.577,A -85,B 0,C 180,E1 -27431.026,E2 -27431.026} C_VEL
LIN {X 0,Y 85.539,Z 726.309,A -85,B 0,C 180,E1 -27440.542,E2 -27440.542} C_VEL
LIN {X 0,Y 85.87,Z 727.077,A -85,B 0,C 180,E1 -27445.306,E2 -27445.306} C_VEL
LIN {X 0,Y 86.612,Z 727.428,A -85,B 0,C 180,E1 -27450,E2 -27450} C_VEL
LIN {X 0,Y 85.879,Z 727.061,A -85,B 0,C 180,E1 -27454.694,E2 -27454.694} C_VEL
LIN {X 0,Y 85.528,Z 726.256,A -85,B 0,C 180,E1 -27459.575,E2 -27459.575} C_VEL
LIN {X 0,Y 86.467,Z 723.521,A -85,B 0,C 180,E1 -27468.972,E2 -27468.972} C_VEL
LIN {X 0,Y 88.773,Z 720.33,A -85,B 0,C 180,E1 -27475.812,E2 -27475.812} C_VEL
LIN {X 0,Y 93.377,Z 715.063,A -85,B 0,C 180,E1 -27483.439,E2 -27483.439} C_VEL
LIN {X 0,Y 98.987,Z 708.716,A -85,B 0,C 180,E1 -27489.716,E2 -27489.716} C_VEL
LIN {X 0,Y 105.032,Z 701.625,A -85,B 0,C 180,E1 -27494.633,E2 -27494.633} C_VEL
LIN {X 0,Y 111.83,Z 692.799,A -85,B 0,C 180,E1 -27498.949,E2 -27498.949} C_VEL
LIN {X 0,Y 118.08,Z 683.825,A -85,B 0,C 180,E1 -27502.056,E2 -27502.056} C_VEL
LIN {X 0,Y 123.381,Z 675.194,A -85,B 0,C 180,E1 -27504.261,E2 -27504.261} C_VEL
LIN {X 0,Y 128.747,Z 664.691,A -85,B 0,C 180,E1 -27506.35,E2 -27506.35} C_VEL
LIN {X 0,Y 133.664,Z 653.064,A -85,B 0,C 180,E1 -27508.024,E2 -27508.024} C_VEL
LIN {X 0,Y 137.564,Z 640.878,A -85,B 0,C 180,E1 -27509.314,E2 -27509.314} C_VEL
LIN {X 0,Y 140.715,Z 627.302,A -85,B 0,C 180,E1 -27510.268,E2 -27510.268} C_VEL
LIN {X 0,Y 141.609,Z 621.203,A -85,B 0,C 180,E1 -27510.641,E2 -27510.641} C_VEL
LIN {X 0,Y 142.324,Z 592.534,A -85,B 0,C 180,E1 -27513.201,E2 -27513.201} C_VEL
LIN {X 0,Y 139.859,Z 583.883,A -85,B 0,C 180,E1 -27516.198,E2 -27516.198} C_VEL
LIN {X 0,Y 139.219,Z 581.925,A -85,B 0,C 180,E1 -27517.016,E2 -27517.016} C_VEL
LIN {X 0,Y 138.286,Z 579.471,A -85,B 0,C 180,E1 -27518.22,E2 -27518.22} C_VEL
LIN {X 0,Y 136.646,Z 576.774,A -85,B 0,C 180,E1 -27520.306,E2 -27520.306} C_VEL
LIN {X 0,Y 133.897,Z 573.848,A -85,B 0,C 180,E1 -27524.207,E2 -27524.207} C_VEL
LIN {X 0,Y 132.117,Z 571.594,A -85,B 0,C 180,E1 -27527.491,E2 -27527.491} C_VEL
LIN {X 0,Y 131.471,Z 570.074,A -85,B 0,C 180,E1 -27529.105,E2 -27529.105} C_VEL
LIN {X 0,Y 130.976,Z 568.173,A -85,B 0,C 180,E1 -27530.737,E2 -27530.737} C_VEL
LIN {X 0,Y 129.407,Z 564.01,A -85,B 0,C 180,E1 -27540,E2 -27540} C_VEL
LIN {X 0,Y 129.397,Z 564.391,A -85,B 0,C 180,E1 -27542.724,E2 -27542.724} C_VEL
LIN {X 0,Y 130.954,Z 568.204,A -85,B 0,C 180,E1 -27551.243,E2 -27551.243} C_VEL
LIN {X 0,Y 133.365,Z 572.837,A -85,B 0,C 180,E1 -27556.848,E2 -27556.848} C_VEL
LIN {X 0,Y 135.423,Z 576.729,A -85,B 0,C 180,E1 -27560.296,E2 -27560.296} C_VEL
LIN {X 0,Y 138.245,Z 582.377,A -85,B 0,C 180,E1 -27564.143,E2 -27564.143} C_VEL
LIN {X 0,Y 141.333,Z 589.389,A -85,B 0,C 180,E1 -27567.705,E2 -27567.705} C_VEL
LIN {X 0,Y 141.65,Z 590.154,A -85,B 0,C 180,E1 -27568.043,E2 -27568.043} C_VEL
LIN {X 0,Y 140.177,Z 605.324,A -85,B 0,C 180,E1 -27568.91,E2 -27568.91} C_VEL
LIN {X 0,Y 137.829,Z 617.705,A -85,B 0,C 180,E1 -27569.909,E2 -27569.909} C_VEL
LIN {X 0,Y 134.199,Z 630.631,A -85,B 0,C 180,E1 -27571.436,E2 -27571.436} C_VEL
LIN {X 0,Y 130.148,Z 641.446,A -85,B 0,C 180,E1 -27573.125,E2 -27573.125} C_VEL
LIN {X 0,Y 125.49,Z 651.22,A -85,B 0,C 180,E1 -27575.01,E2 -27575.01} C_VEL
LIN {X 0,Y 120.457,Z 660.253,A -85,B 0,C 180,E1 -27577.352,E2 -27577.352} C_VEL
LIN {X 0,Y 115.042,Z 668.651,A -85,B 0,C 180,E1 -27580.216,E2 -27580.216} C_VEL
LIN {X 0,Y 109.363,Z 676.367,A -85,B 0,C 180,E1 -27583.702,E2 -27583.702} C_VEL
LIN {X 0,Y 102.823,Z 684.022,A -85,B 0,C 180,E1 -27588.341,E2 -27588.341} C_VEL
LIN {X 0,Y 96.265,Z 690.815,A -85,B 0,C 180,E1 -27594.265,E2 -27594.265} C_VEL
LIN {X 0,Y 91.266,Z 695.416,A -85,B 0,C 180,E1 -27599.965,E2 -27599.965} C_VEL
LIN {X 0,Y 87,Z 698.951,A -85,B 0,C 180,E1 -27606.178,E2 -27606.178} C_VEL
LIN {X 0,Y 84.729,Z 700.77,A -85,B 0,C 180,E1 -27610.623,E2 -27610.623} C_VEL
LIN {X 0,Y 82.055,Z 703.043,A -85,B 0,C 180,E1 -27620.137,E2 -27620.137} C_VEL
LIN {X 0,Y 80.972,Z 703.865,A -85,B 0,C 180,E1 -27630,E2 -27630} C_VEL
LIN {X 0,Y 82.051,Z 703.087,A -85,B 0,C 180,E1 -27639.864,E2 -27639.864} C_VEL
LIN {X 0,Y 84.71,Z 700.86,A -85,B 0,C 180,E1 -27649.381,E2 -27649.381} C_VEL
LIN {X 0,Y 88.372,Z 698.02,A -85,B 0,C 180,E1 -27655.937,E2 -27655.937} C_VEL
LIN {X 0,Y 92.895,Z 694.183,A -85,B 0,C 180,E1 -27661.977,E2 -27661.977} C_VEL
LIN {X 0,Y 98.181,Z 689.09,A -85,B 0,C 180,E1 -27667.734,E2 -27667.734} C_VEL
LIN {X 0,Y 103.934,Z 683.044,A -85,B 0,C 180,E1 -27672.546,E2 -27672.546} C_VEL
LIN {X 0,Y 110.464,Z 675.25,A -85,B 0,C 180,E1 -27677.024,E2 -27677.024} C_VEL
LIN {X 0,Y 117.378,Z 665.562,A -85,B 0,C 180,E1 -27681.11,E2 -27681.11} C_VEL
LIN {X 0,Y 122.904,Z 656.493,A -85,B 0,C 180,E1 -27683.871,E2 -27683.871} C_VEL
LIN {X 0,Y 128.867,Z 644.921,A -85,B 0,C 180,E1 -27686.395,E2 -27686.395} C_VEL
LIN {X 0,Y 133.709,Z 632.94,A -85,B 0,C 180,E1 -27688.388,E2 -27688.388} C_VEL
LIN {X 0,Y 137.59,Z 620.265,A -85,B 0,C 180,E1 -27689.862,E2 -27689.862} C_VEL
LIN {X 0,Y 140.112,Z 607.579,A -85,B 0,C 180,E1 -27691.064,E2 -27691.064} C_VEL
LIN {X 0,Y 141.542,Z 595.38,A -85,B 0,C 180,E1 -27691.823,E2 -27691.823} C_VEL
LIN {X 0,Y 141.865,Z 590.315,A -85,B 0,C 180,E1 -27692.12,E2 -27692.12} C_VEL
LIN {X 0,Y 138.781,Z 583.24,A -85,B 0,C 180,E1 -27695.635,E2 -27695.635} C_VEL
LIN {X 0,Y 135.619,Z 576.718,A -85,B 0,C 180,E1 -27699.953,E2 -27699.953} C_VEL
LIN {X 0,Y 133.022,Z 571.923,A -85,B 0,C 180,E1 -27704.486,E2 -27704.486} C_VEL
LIN {X 0,Y 131.135,Z 568.282,A -85,B 0,C 180,E1 -27709.188,E2 -27709.188} C_VEL
LIN {X 0,Y 129.671,Z 564.534,A -85,B 0,C 180,E1 -27718.447,E2 -27718.447} C_VEL
LIN {X 0,Y 129.672,Z 564.852,A -85,B 0,C 180,E1 -27720.582,E2 -27720.582} C_VEL
LIN {X 0,Y 131.255,Z 568.504,A -85,B 0,C 180,E1 -27729.244,E2 -27729.244} C_VEL
LIN {X 0,Y 132.999,Z 574.081,A -85,B 0,C 180,E1 -27733.993,E2 -27733.993} C_VEL
LIN {X 0,Y 134.611,Z 579.246,A -85,B 0,C 180,E1 -27737.26,E2 -27737.26} C_VEL
LIN {X 0,Y 136.615,Z 585.913,A -85,B 0,C 180,E1 -27740.614,E2 -27740.614} C_VEL
LIN {X 0,Y 139.084,Z 595.004,A -85,B 0,C 180,E1 -27744.16,E2 -27744.16} C_VEL
LIN {X 0,Y 139.241,Z 596.724,A -85,B 0,C 180,E1 -27744.501,E2 -27744.501} C_VEL
LIN {X 0,Y 138.366,Z 620.638,A -85,B 0,C 180,E1 -27746.693,E2 -27746.693} C_VEL
LIN {X 0,Y 137.38,Z 627.176,A -85,B 0,C 180,E1 -27747.129,E2 -27747.129} C_VEL
LIN {X 0,Y 134.532,Z 639.147,A -85,B 0,C 180,E1 -27747.954,E2 -27747.954} C_VEL
LIN {X 0,Y 130.572,Z 651.13,A -85,B 0,C 180,E1 -27749.11,E2 -27749.11} C_VEL
LIN {X 0,Y 125.678,Z 662.712,A -85,B 0,C 180,E1 -27750.71,E2 -27750.71} C_VEL
LIN {X 0,Y 119.307,Z 674.552,A -85,B 0,C 180,E1 -27752.923,E2 -27752.923} C_VEL
LIN {X 0,Y 112.505,Z 685.096,A -85,B 0,C 180,E1 -27755.702,E2 -27755.702} C_VEL
LIN {X 0,Y 106.022,Z 693.654,A -85,B 0,C 180,E1 -27758.843,E2 -27758.843} C_VEL
LIN {X 0,Y 98.919,Z 702.071,A -85,B 0,C 180,E1 -27763.263,E2 -27763.263} C_VEL
LIN {X 0,Y 92.602,Z 708.908,A -85,B 0,C 180,E1 -27768.39,E2 -27768.39} C_VEL
LIN {X 0,Y 88.269,Z 713.416,A -85,B 0,C 180,E1 -27773.052,E2 -27773.052} C_VEL
LIN {X 0,Y 83.547,Z 718.103,A -85,B 0,C 180,E1 -27779.688,E2 -27779.688} C_VEL
LIN {X 0,Y 80.432,Z 721.598,A -85,B 0,C 180,E1 -27786.847,E2 -27786.847} C_VEL
LIN {X 0,Y 78.761,Z 724.131,A -85,B 0,C 180,E1 -27794.473,E2 -27794.473} C_VEL
LIN {X 0,Y 78.491,Z 725.37,A -85,B 0,C 180,E1 -27800.039,E2 -27800.039} C_VEL
LIN {X 0,Y 78.772,Z 726.076,A -85,B 0,C 180,E1 -27804.881,E2 -27804.881} C_VEL
LIN {X 0,Y 79.501,Z 726.429,A -85,B 0,C 180,E1 -27810,E2 -27810} C_VEL
LIN {X 0,Y 78.779,Z 726.059,A -85,B 0,C 180,E1 -27815.118,E2 -27815.118} C_VEL
LIN {X 0,Y 78.479,Z 725.273,A -85,B 0,C 180,E1 -27820.317,E2 -27820.317} C_VEL
LIN {X 0,Y 79.719,Z 722.512,A -85,B 0,C 180,E1 -27830.648,E2 -27830.648} C_VEL
LIN {X 0,Y 82.383,Z 719.322,A -85,B 0,C 180,E1 -27837.981,E2 -27837.981} C_VEL
LIN {X 0,Y 86.459,Z 715.122,A -85,B 0,C 180,E1 -27844.68,E2 -27844.68} C_VEL
LIN {X 0,Y 92.602,Z 708.75,A -85,B 0,C 180,E1 -27851.61,E2 -27851.61} C_VEL
LIN {X 0,Y 98.926,Z 701.879,A -85,B 0,C 180,E1 -27856.733,E2 -27856.733} C_VEL
LIN {X 0,Y 106.037,Z 693.422,A -85,B 0,C 180,E1 -27861.147,E2 -27861.147} C_VEL
LIN {X 0,Y 112.51,Z 684.795,A -85,B 0,C 180,E1 -27864.295,E2 -27864.295} C_VEL
LIN {X 0,Y 118.682,Z 675.377,A -85,B 0,C 180,E1 -27866.764,E2 -27866.764} C_VEL
LIN {X 0,Y 124.238,Z 665.124,A -85,B 0,C 180,E1 -27868.824,E2 -27868.824} C_VEL
LIN {X 0,Y 129.257,Z 653.966,A -85,B 0,C 180,E1 -27870.451,E2 -27870.451} C_VEL
LIN {X 0,Y 133.508,Z 641.834,A -85,B 0,C 180,E1 -27871.762,E2 -27871.762} C_VEL
LIN {X 0,Y 136.759,Z 629.072,A -85,B 0,C 180,E1 -27872.698,E2 -27872.698} C_VEL
LIN {X 0,Y 137.935,Z 622.585,A -85,B 0,C 180,E1 -27873.058,E2 -27873.058} C_VEL
LIN {X 0,Y 138.839,Z 603,A -85,B 0,C 180,E1 -27874.835,E2 -27874.835} C_VEL
LIN {X 0,Y 138.935,Z 595.252,A -85,B 0,C 180,E1 -27875.656,E2 -27875.656} C_VEL
LIN {X 0,Y 136.766,Z 587.157,A -85,B 0,C 180,E1 -27878.72,E2 -27878.72} C_VEL
LIN {X 0,Y 134.76,Z 580.361,A -85,B 0,C 180,E1 -27881.962,E2 -27881.962} C_VEL
LIN {X 0,Y 133.441,Z 576.139,A -85,B 0,C 180,E1 -27884.438,E2 -27884.438} C_VEL
LIN {X 0,Y 132.191,Z 572.146,A -85,B 0,C 180,E1 -27887.234,E2 -27887.234} C_VEL
LIN {X 0,Y 131.471,Z 570.074,A -85,B 0,C 180,E1 -27889.105,E2 -27889.105} C_VEL
LIN {X 0,Y 130.911,Z 568.78,A -85,B 0,C 180,E1 -27890.711,E2 -27890.711} C_VEL
LIN {X 0,Y 130.076,Z 568.051,A -85,B 0,C 180,E1 -27893.27,E2 -27893.27} C_VEL
LIN {X 0,Y 129.364,Z 568.402,A -85,B 0,C 180,E1 -27895.887,E2 -27895.887} C_VEL
LIN {X 0,Y 128.52,Z 571.739,A -85,B 0,C 180,E1 -27903.064,E2 -27903.064} C_VEL
LIN {X 0,Y 130.067,Z 575.564,A -85,B 0,C 180,E1 -27911.32,E2 -27911.32} C_VEL
LIN {X 0,Y 132.032,Z 579.68,A -85,B 0,C 180,E1 -27916.129,E2 -27916.129} C_VEL
LIN {X 0,Y 133.885,Z 583.438,A -85,B 0,C 180,E1 -27919.465,E2 -27919.465} C_VEL
LIN {X 0,Y 136.596,Z 589.431,A -85,B 0,C 180,E1 -27923.439,E2 -27923.439} C_VEL
LIN {X 0,Y 138.276,Z 593.592,A -85,B 0,C 180,E1 -27925.583,E2 -27925.583} C_VEL
LIN {X 0,Y 136.806,Z 607.004,A -85,B 0,C 180,E1 -27926.363,E2 -27926.363} C_VEL
LIN {X 0,Y 134.459,Z 618.703,A -85,B 0,C 180,E1 -27927.309,E2 -27927.309} C_VEL
LIN {X 0,Y 130.964,Z 630.799,A -85,B 0,C 180,E1 -27928.702,E2 -27928.702} C_VEL
LIN {X 0,Y 126.737,Z 641.757,A -85,B 0,C 180,E1 -27930.338,E2 -27930.338} C_VEL
LIN {X 0,Y 121.595,Z 652.212,A -85,B 0,C 180,E1 -27932.298,E2 -27932.298} C_VEL
LIN {X 0,Y 116.327,Z 661.245,A -85,B 0,C 180,E1 -27934.599,E2 -27934.599} C_VEL
LIN {X 0,Y 110.634,Z 669.642,A -85,B 0,C 180,E1 -27937.436,E2 -27937.436} C_VEL
LIN {X 0,Y 104.631,Z 677.357,A -85,B 0,C 180,E1 -27940.919,E2 -27940.919} C_VEL
LIN {X 0,Y 97.684,Z 685.012,A -85,B 0,C 180,E1 -27945.6,E2 -27945.6} C_VEL
LIN {X 0,Y 90.653,Z 691.805,A -85,B 0,C 180,E1 -27951.669,E2 -27951.669} C_VEL
LIN {X 0,Y 85.254,Z 696.406,A -85,B 0,C 180,E1 -27957.601,E2 -27957.601} C_VEL
LIN {X 0,Y 80.619,Z 699.94,A -85,B 0,C 180,E1 -27964.16,E2 -27964.16} C_VEL
LIN {X 0,Y 78.132,Z 701.76,A -85,B 0,C 180,E1 -27968.913,E2 -27968.913} C_VEL
LIN {X 0,Y 75.14,Z 704.032,A -85,B 0,C 180,E1 -27979.219,E2 -27979.219} C_VEL
LIN {X 0,Y 73.944,Z 704.853,A -85,B 0,C 180,E1 -27990,E2 -27990} C_VEL
LIN {X 0,Y 75.137,Z 704.075,A -85,B 0,C 180,E1 -28000.782,E2 -28000.782} C_VEL
LIN {X 0,Y 78.113,Z 701.848,A -85,B 0,C 180,E1 -28011.093,E2 -28011.093} C_VEL
LIN {X 0,Y 82.109,Z 699.008,A -85,B 0,C 180,E1 -28018.083,E2 -28018.083} C_VEL
LIN {X 0,Y 87.013,Z 695.17,A -85,B 0,C 180,E1 -28024.428,E2 -28024.428} C_VEL
LIN {X 0,Y 92.722,Z 690.077,A -85,B 0,C 180,E1 -28030.392,E2 -28030.392} C_VEL
LIN {X 0,Y 98.87,Z 684.03,A -85,B 0,C 180,E1 -28035.301,E2 -28035.301} C_VEL
LIN {X 0,Y 105.798,Z 676.236,A -85,B 0,C 180,E1 -28039.81,E2 -28039.81} C_VEL
LIN {X 0,Y 113.097,Z 666.548,A -85,B 0,C 180,E1 -28043.883,E2 -28043.883} C_VEL
LIN {X 0,Y 118.896,Z 657.477,A -85,B 0,C 180,E1 -28046.607,E2 -28046.607} C_VEL
LIN {X 0,Y 125.108,Z 645.906,A -85,B 0,C 180,E1 -28049.081,E2 -28049.081} C_VEL
LIN {X 0,Y 130.164,Z 633.921,A -85,B 0,C 180,E1 -28051.022,E2 -28051.022} C_VEL
LIN {X 0,Y 133.823,Z 622.659,A -85,B 0,C 180,E1 -28052.319,E2 -28052.319} C_VEL
LIN {X 0,Y 136.688,Z 609.457,A -85,B 0,C 180,E1 -28053.571,E2 -28053.571} C_VEL
LIN {X 0,Y 138.323,Z 596.603,A -85,B 0,C 180,E1 -28054.392,E2 -28054.392} C_VEL
LIN {X 0,Y 138.528,Z 593.826,A -85,B 0,C 180,E1 -28054.547,E2 -28054.547} C_VEL
LIN {X 0,Y 135.729,Z 587.078,A -85,B 0,C 180,E1 -28058.25,E2 -28058.25} C_VEL
LIN {X 0,Y 133.393,Z 582.002,A -85,B 0,C 180,E1 -28061.969,E2 -28061.969} C_VEL
LIN {X 0,Y 131.497,Z 578.312,A -85,B 0,C 180,E1 -28065.738,E2 -28065.738} C_VEL
LIN {X 0,Y 130.019,Z 575.12,A -85,B 0,C 180,E1 -28069.882,E2 -28069.882} C_VEL
LIN {X 0,Y 128.793,Z 571.683,A -85,B 0,C 180,E1 -28078.436,E2 -28078.436} C_VEL
LIN {X 0,Y 128.793,Z 572.015,A -85,B 0,C 180,E1 -28080.586,E2 -28080.586} C_VEL
LIN {X 0,Y 130.059,Z 575.291,A -85,B 0,C 180,E1 -28088.35,E2 -28088.35} C_VEL
LIN {X 0,Y 131.418,Z 580.261,A -85,B 0,C 180,E1 -28092.634,E2 -28092.634} C_VEL
LIN {X 0,Y 132.784,Z 585.305,A -85,B 0,C 180,E1 -28095.837,E2 -28095.837} C_VEL
LIN {X 0,Y 134.465,Z 591.695,A -85,B 0,C 180,E1 -28099.066,E2 -28099.066} C_VEL
LIN {X 0,Y 136.211,Z 598.967,A -85,B 0,C 180,E1 -28101.976,E2 -28101.976} C_VEL
LIN {X 0,Y 135.229,Z 619.633,A -85,B 0,C 180,E1 -28103.917,E2 -28103.917} C_VEL
LIN {X 0,Y 134.386,Z 625.682,A -85,B 0,C 180,E1 -28104.396,E2 -28104.396} C_VEL
LIN {X 0,Y 131.245,Z 638.512,A -85,B 0,C 180,E1 -28105.24,E2 -28105.24} C_VEL
LIN {X 0,Y 126.704,Z 651.575,A -85,B 0,C 180,E1 -28106.476,E2 -28106.476} C_VEL
LIN {X 0,Y 121.458,Z 663.153,A -85,B 0,C 180,E1 -28108.067,E2 -28108.067} C_VEL
LIN {X 0,Y 114.871,Z 674.74,A -85,B 0,C 180,E1 -28110.212,E2 -28110.212} C_VEL
LIN {X 0,Y 108.51,Z 684.099,A -85,B 0,C 180,E1 -28112.652,E2 -28112.652} C_VEL
LIN {X 0,Y 101.709,Z 692.656,A -85,B 0,C 180,E1 -28115.718,E2 -28115.718} C_VEL
LIN {X 0,Y 94.181,Z 701.072,A -85,B 0,C 180,E1 -28120.106,E2 -28120.106} C_VEL
LIN {X 0,Y 87.402,Z 707.908,A -85,B 0,C 180,E1 -28125.286,E2 -28125.286} C_VEL
LIN {X 0,Y 80.678,Z 714.23,A -85,B 0,C 180,E1 -28132.427,E2 -28132.427} C_VEL
LIN {X 0,Y 76.103,Z 718.394,A -85,B 0,C 180,E1 -28139.476,E2 -28139.476} C_VEL
LIN {X 0,Y 73.03,Z 721.559,A -85,B 0,C 180,E1 -28147.361,E2 -28147.361} C_VEL
LIN {X 0,Y 71.444,Z 724.295,A -85,B 0,C 180,E1 -28158.654,E2 -28158.654} C_VEL
LIN {X 0,Y 71.657,Z 725.071,A -85,B 0,C 180,E1 -28164.372,E2 -28164.372} C_VEL
LIN {X 0,Y 72.389,Z 725.428,A -85,B 0,C 180,E1 -28170,E2 -28170} C_VEL
LIN {X 0,Y 71.427,Z 724.447,A -85,B 0,C 180,E1 -28180.284,E2 -28180.284} C_VEL
LIN {X 0,Y 71.885,Z 723.084,A -85,B 0,C 180,E1 -28187.055,E2 -28187.055} C_VEL
LIN {X 0,Y 73.898,Z 720.524,A -85,B 0,C 180,E1 -28195.338,E2 -28195.338} C_VEL
LIN {X 0,Y 77.506,Z 717.008,A -85,B 0,C 180,E1 -28202.96,E2 -28202.96} C_VEL
LIN {X 0,Y 82.935,Z 711.995,A -85,B 0,C 180,E1 -28210.3,E2 -28210.3} C_VEL
LIN {X 0,Y 89.544,Z 705.635,A -85,B 0,C 180,E1 -28216.551,E2 -28216.551} C_VEL
LIN {X 0,Y 96.633,Z 698.251,A -85,B 0,C 180,E1 -28221.427,E2 -28221.427} C_VEL
LIN {X 0,Y 104.39,Z 689.143,A -85,B 0,C 180,E1 -28225.558,E2 -28225.558} C_VEL
LIN {X 0,Y 111.353,Z 679.847,A -85,B 0,C 180,E1 -28228.433,E2 -28228.433} C_VEL
LIN {X 0,Y 117.768,Z 669.502,A -85,B 0,C 180,E1 -28230.78,E2 -28230.78} C_VEL
LIN {X 0,Y 123.66,Z 658.069,A -85,B 0,C 180,E1 -28232.622,E2 -28232.622} C_VEL
LIN {X 0,Y 128.183,Z 647.02,A -85,B 0,C 180,E1 -28233.946,E2 -28233.946} C_VEL
LIN {X 0,Y 132.185,Z 634.322,A -85,B 0,C 180,E1 -28234.997,E2 -28234.997} C_VEL
LIN {X 0,Y 134.674,Z 622.377,A -85,B 0,C 180,E1 -28235.766,E2 -28235.766} C_VEL
LIN {X 0,Y 135.76,Z 604.354,A -85,B 0,C 180,E1 -28237.441,E2 -28237.441} C_VEL
LIN {X 0,Y 135.92,Z 598.643,A -85,B 0,C 180,E1 -28238.033,E2 -28238.033} C_VEL
LIN {X 0,Y 134.005,Z 590.595,A -85,B 0,C 180,E1 -28241.263,E2 -28241.263} C_VEL
LIN {X 0,Y 132.082,Z 583.314,A -85,B 0,C 180,E1 -28245.093,E2 -28245.093} C_VEL
LIN {X 0,Y 130.722,Z 578.498,A -85,B 0,C 180,E1 -28248.48,E2 -28248.48} C_VEL
LIN {X 0,Y 129.719,Z 574.859,A -85,B 0,C 180,E1 -28251.824,E2 -28251.824} C_VEL
LIN {X 0,Y 128.522,Z 571.215,A -85,B 0,C 180,E1 -28260,E2 -28260} C_VEL
LIN {X 0,Y 128.513,Z 571.408,A -85,B 0,C 180,E1 -28262.351,E2 -28262.351} C_VEL
LIN {X 0,Y 128.52,Z 571.739,A -85,B 0,C 180,E1 -28263.064,E2 -28263.064} C_VEL
LIN {X 0,Y 128.618,Z 573.58,A -85,B 0,C 180,E1 -28265.571,E2 -28265.571} C_VEL
LIN {X 0,Y 129.003,Z 578.427,A -85,B 0,C 180,E1 -28269.421,E2 -28269.421} C_VEL
LIN {X 0,Y 130.109,Z 584.86,A -85,B 0,C 180,E1 -28273.91,E2 -28273.91} C_VEL
LIN {X 0,Y 130.749,Z 586.628,A -85,B 0,C 180,E1 -28275.467,E2 -28275.467} C_VEL
LIN {X 0,Y 132.619,Z 590.719,A -85,B 0,C 180,E1 -28279.041,E2 -28279.041} C_VEL
LIN {X 0,Y 135.061,Z 596.889,A -85,B 0,C 180,E1 -28282.872,E2 -28282.872} C_VEL
LIN {X 0,Y 135.184,Z 597.251,A -85,B 0,C 180,E1 -28283.052,E2 -28283.052} C_VEL
LIN {X 0,Y 133.378,Z 610.564,A -85,B 0,C 180,E1 -28283.857,E2 -28283.857} C_VEL
LIN {X 0,Y 130.238,Z 623.945,A -85,B 0,C 180,E1 -28285.015,E2 -28285.015} C_VEL
LIN {X 0,Y 126.215,Z 635.887,A -85,B 0,C 180,E1 -28286.453,E2 -28286.453} C_VEL
LIN {X 0,Y 121.167,Z 647.222,A -85,B 0,C 180,E1 -28288.247,E2 -28288.247} C_VEL
LIN {X 0,Y 115.217,Z 657.942,A -85,B 0,C 180,E1 -28290.506,E2 -28290.506} C_VEL
LIN {X 0,Y 109.137,Z 667.114,A -85,B 0,C 180,E1 -28293.162,E2 -28293.162} C_VEL
LIN {X 0,Y 102.683,Z 675.444,A -85,B 0,C 180,E1 -28296.468,E2 -28296.468} C_VEL
LIN {X 0,Y 95.28,Z 683.541,A -85,B 0,C 180,E1 -28300.884,E2 -28300.884} C_VEL
LIN {X 0,Y 87.744,Z 690.638,A -85,B 0,C 180,E1 -28306.447,E2 -28306.447} C_VEL
LIN {X 0,Y 81.334,Z 695.996,A -85,B 0,C 180,E1 -28312.782,E2 -28312.782} C_VEL
LIN {X 0,Y 75.988,Z 699.877,A -85,B 0,C 180,E1 -28319.424,E2 -28319.424} C_VEL
LIN {X 0,Y 71.617,Z 702.749,A -85,B 0,C 180,E1 -28326.888,E2 -28326.888} C_VEL
LIN {X 0,Y 68.248,Z 705.02,A -85,B 0,C 180,E1 -28338.115,E2 -28338.115} C_VEL
LIN {X 0,Y 66.916,Z 705.842,A -85,B 0,C 180,E1 -28350,E2 -28350} C_VEL
LIN {X 0,Y 68.245,Z 705.063,A -85,B 0,C 180,E1 -28361.886,E2 -28361.886} C_VEL
LIN {X 0,Y 71.598,Z 702.836,A -85,B 0,C 180,E1 -28373.118,E2 -28373.118} C_VEL
LIN {X 0,Y 75.981,Z 699.995,A -85,B 0,C 180,E1 -28380.579,E2 -28380.579} C_VEL
LIN {X 0,Y 81.313,Z 696.157,A -85,B 0,C 180,E1 -28387.229,E2 -28387.229} C_VEL
LIN {X 0,Y 87.488,Z 691.064,A -85,B 0,C 180,E1 -28393.376,E2 -28393.376} C_VEL
LIN {X 0,Y 94.06,Z 685.017,A -85,B 0,C 180,E1 -28398.346,E2 -28398.346} C_VEL
LIN {X 0,Y 101.404,Z 677.221,A -85,B 0,C 180,E1 -28402.845,E2 -28402.845} C_VEL
LIN {X 0,Y 109.102,Z 667.533,A -85,B 0,C 180,E1 -28406.867,E2 -28406.867} C_VEL
LIN {X 0,Y 115.177,Z 658.462,A -85,B 0,C 180,E1 -28409.527,E2 -28409.527} C_VEL
LIN {X 0,Y 121.651,Z 646.89,A -85,B 0,C 180,E1 -28411.917,E2 -28411.917} C_VEL
LIN {X 0,Y 126.852,Z 635.041,A -85,B 0,C 180,E1 -28413.785,E2 -28413.785} C_VEL
LIN {X 0,Y 130.942,Z 622.762,A -85,B 0,C 180,E1 -28415.138,E2 -28415.138} C_VEL
LIN {X 0,Y 133.864,Z 609.594,A -85,B 0,C 180,E1 -28416.334,E2 -28416.334} C_VEL
LIN {X 0,Y 135.375,Z 597.271,A -85,B 0,C 180,E1 -28417.179,E2 -28417.179} C_VEL
LIN {X 0,Y 132.917,Z 591.087,A -85,B 0,C 180,E1 -28421.023,E2 -28421.023} C_VEL
LIN {X 0,Y 131.482,Z 587.839,A -85,B 0,C 180,E1 -28423.702,E2 -28423.702} C_VEL
LIN {X 0,Y 130.139,Z 584.902,A -85,B 0,C 180,E1 -28426.757,E2 -28426.757} C_VEL
LIN {X 0,Y 128.92,Z 581.985,A -85,B 0,C 180,E1 -28430.587,E2 -28430.587} C_VEL
LIN {X 0,Y 127.918,Z 578.814,A -85,B 0,C 180,E1 -28438.426,E2 -28438.426} C_VEL
LIN {X 0,Y 127.912,Z 579.189,A -85,B 0,C 180,E1 -28440.59,E2 -28440.59} C_VEL
LIN {X 0,Y 128.895,Z 582.081,A -85,B 0,C 180,E1 -28447.44,E2 -28447.44} C_VEL
LIN {X 0,Y 129.87,Z 586.286,A -85,B 0,C 180,E1 -28451.115,E2 -28451.115} C_VEL
LIN {X 0,Y 131.094,Z 591.578,A -85,B 0,C 180,E1 -28454.505,E2 -28454.505} C_VEL
LIN {X 0,Y 132.548,Z 598.114,A -85,B 0,C 180,E1 -28457.747,E2 -28457.747} C_VEL
LIN {X 0,Y 133.412,Z 602.294,A -85,B 0,C 180,E1 -28459.454,E2 -28459.454} C_VEL
LIN {X 0,Y 132.236,Z 620.218,A -85,B 0,C 180,E1 -28461.165,E2 -28461.165} C_VEL
LIN {X 0,Y 131.415,Z 625.597,A -85,B 0,C 180,E1 -28461.618,E2 -28461.618} C_VEL
LIN {X 0,Y 127.906,Z 639.06,A -85,B 0,C 180,E1 -28462.47,E2 -28462.47} C_VEL
LIN {X 0,Y 123.683,Z 650.576,A -85,B 0,C 180,E1 -28463.51,E2 -28463.51} C_VEL
LIN {X 0,Y 118.276,Z 662.156,A -85,B 0,C 180,E1 -28465.023,E2 -28465.023} C_VEL
LIN {X 0,Y 111.457,Z 673.742,A -85,B 0,C 180,E1 -28467.046,E2 -28467.046} C_VEL
LIN {X 0,Y 104.849,Z 683.104,A -85,B 0,C 180,E1 -28469.382,E2 -28469.382} C_VEL
LIN {X 0,Y 96.345,Z 693.168,A -85,B 0,C 180,E1 -28472.98,E2 -28472.98} C_VEL
LIN {X 0,Y 88.485,Z 701.333,A -85,B 0,C 180,E1 -28477.416,E2 -28477.416} C_VEL
LIN {X 0,Y 81.343,Z 707.929,A -85,B 0,C 180,E1 -28482.745,E2 -28482.745} C_VEL
LIN {X 0,Y 75.158,Z 713.23,A -85,B 0,C 180,E1 -28489.114,E2 -28489.114} C_VEL
LIN {X 0,Y 70.024,Z 717.387,A -85,B 0,C 180,E1 -28496.496,E2 -28496.496} C_VEL
LIN {X 0,Y 66.462,Z 720.551,A -85,B 0,C 180,E1 -28504.978,E2 -28504.978} C_VEL
LIN {X 0,Y 64.429,Z 723.287,A -85,B 0,C 180,E1 -28517.399,E2 -28517.399} C_VEL
LIN {X 0,Y 64.549,Z 724.067,A -85,B 0,C 180,E1 -28523.75,E2 -28523.75} C_VEL
LIN {X 0,Y 65.275,Z 724.428,A -85,B 0,C 180,E1 -28530,E2 -28530} C_VEL
LIN {X 0,Y 64.394,Z 723.535,A -85,B 0,C 180,E1 -28540.807,E2 -28540.807} C_VEL
LIN {X 0,Y 65.057,Z 722.074,A -85,B 0,C 180,E1 -28548.91,E2 -28548.91} C_VEL
LIN {X 0,Y 67.487,Z 719.515,A -85,B 0,C 180,E1 -28557.944,E2 -28557.944} C_VEL
LIN {X 0,Y 71.602,Z 716,A -85,B 0,C 180,E1 -28566.08,E2 -28566.08} C_VEL
LIN {X 0,Y 77.158,Z 711.373,A -85,B 0,C 180,E1 -28573.224,E2 -28573.224} C_VEL
LIN {X 0,Y 84.789,Z 704.629,A -85,B 0,C 180,E1 -28580.058,E2 -28580.058} C_VEL
LIN {X 0,Y 92.35,Z 697.245,A -85,B 0,C 180,E1 -28584.892,E2 -28584.892} C_VEL
LIN {X 0,Y 100.546,Z 688.142,A -85,B 0,C 180,E1 -28588.896,E2 -28588.896} C_VEL
LIN {X 0,Y 107.814,Z 678.848,A -85,B 0,C 180,E1 -28591.641,E2 -28591.641} C_VEL
LIN {X 0,Y 114.469,Z 668.5,A -85,B 0,C 180,E1 -28593.884,E2 -28593.884} C_VEL
LIN {X 0,Y 120.551,Z 657.062,A -85,B 0,C 180,E1 -28595.629,E2 -28595.629} C_VEL
LIN {X 0,Y 125.467,Z 645.382,A -85,B 0,C 180,E1 -28596.932,E2 -28596.932} C_VEL
LIN {X 0,Y 129.572,Z 632.438,A -85,B 0,C 180,E1 -28597.896,E2 -28597.896} C_VEL
LIN {X 0,Y 131.579,Z 623.37,A -85,B 0,C 180,E1 -28598.471,E2 -28598.471} C_VEL
LIN {X 0,Y 132.822,Z 608.76,A -85,B 0,C 180,E1 -28599.883,E2 -28599.883} C_VEL
LIN {X 0,Y 133.105,Z 601.69,A -85,B 0,C 180,E1 -28600.617,E2 -28600.617} C_VEL
LIN {X 0,Y 131.366,Z 593.693,A -85,B 0,C 180,E1 -28604.186,E2 -28604.186} C_VEL
LIN {X 0,Y 130.04,Z 587.938,A -85,B 0,C 180,E1 -28607.515,E2 -28607.515} C_VEL
LIN {X 0,Y 129.241,Z 584.516,A -85,B 0,C 180,E1 -28610.018,E2 -28610.018} C_VEL
LIN {X 0,Y 128.51,Z 581.544,A -85,B 0,C 180,E1 -28612.932,E2 -28612.932} C_VEL
LIN {X 0,Y 127.642,Z 578.38,A -85,B 0,C 180,E1 -28620,E2 -28620} C_VEL
LIN {X 0,Y 127.635,Z 578.425,A -85,B 0,C 180,E1 -28621.972,E2 -28621.972} C_VEL
LIN {X 0,Y 128.898,Z 582.366,A -85,B 0,C 180,E1 -28630.505,E2 -28630.505} C_VEL
LIN {X 0,Y 130.632,Z 586.345,A -85,B 0,C 180,E1 -28635.205,E2 -28635.205} C_VEL
LIN {X 0,Y 130.749,Z 586.628,A -85,B 0,C 180,E1 -28635.467,E2 -28635.467} C_VEL
LIN {X 0,Y 131.431,Z 588.774,A -85,B 0,C 180,E1 -28636.968,E2 -28636.968} C_VEL
LIN {X 0,Y 132.08,Z 592.796,A -85,B 0,C 180,E1 -28638.578,E2 -28638.578} C_VEL
LIN {X 0,Y 132.337,Z 597.663,A -85,B 0,C 180,E1 -28639.756,E2 -28639.756} C_VEL
LIN {X 0,Y 132.071,Z 602.994,A -85,B 0,C 180,E1 -28640.485,E2 -28640.485} C_VEL
LIN {X 0,Y 131.901,Z 604.364,A -85,B 0,C 180,E1 -28640.589,E2 -28640.589} C_VEL
LIN {X 0,Y 129.46,Z 617.343,A -85,B 0,C 180,E1 -28641.485,E2 -28641.485} C_VEL
LIN {X 0,Y 125.94,Z 629.642,A -85,B 0,C 180,E1 -28642.672,E2 -28642.672} C_VEL
LIN {X 0,Y 121.158,Z 641.791,A -85,B 0,C 180,E1 -28644.231,E2 -28644.231} C_VEL
LIN {X 0,Y 115.426,Z 652.926,A -85,B 0,C 180,E1 -28646.095,E2 -28646.095} C_VEL
LIN {X 0,Y 108.96,Z 663.229,A -85,B 0,C 180,E1 -28648.502,E2 -28648.502} C_VEL
LIN {X 0,Y 102.698,Z 671.624,A -85,B 0,C 180,E1 -28651.196,E2 -28651.196} C_VEL
LIN {X 0,Y 96.013,Z 679.339,A -85,B 0,C 180,E1 -28654.567,E2 -28654.567} C_VEL
LIN {X 0,Y 88.191,Z 686.991,A -85,B 0,C 180,E1 -28659.198,E2 -28659.198} C_VEL
LIN {X 0,Y 80.102,Z 693.784,A -85,B 0,C 180,E1 -28665.422,E2 -28665.422} C_VEL
LIN {X 0,Y 73.772,Z 698.384,A -85,B 0,C 180,E1 -28671.741,E2 -28671.741} C_VEL
LIN {X 0,Y 68.241,Z 701.919,A -85,B 0,C 180,E1 -28679.007,E2 -28679.007} C_VEL
LIN {X 0,Y 65.209,Z 703.738,A -85,B 0,C 180,E1 -28684.463,E2 -28684.463} C_VEL
LIN {X 0,Y 61.388,Z 706.009,A -85,B 0,C 180,E1 -28696.764,E2 -28696.764} C_VEL
LIN {X 0,Y 59.888,Z 706.83,A -85,B 0,C 180,E1 -28710,E2 -28710} C_VEL
LIN {X 0,Y 61.384,Z 706.05,A -85,B 0,C 180,E1 -28723.237,E2 -28723.237} C_VEL
LIN {X 0,Y 65.191,Z 703.824,A -85,B 0,C 180,E1 -28735.545,E2 -28735.545} C_VEL
LIN {X 0,Y 70.022,Z 700.982,A -85,B 0,C 180,E1 -28743.505,E2 -28743.505} C_VEL
LIN {X 0,Y 75.837,Z 697.144,A -85,B 0,C 180,E1 -28750.443,E2 -28750.443} C_VEL
LIN {X 0,Y 82.521,Z 692.05,A -85,B 0,C 180,E1 -28756.729,E2 -28756.729} C_VEL
LIN {X 0,Y 89.543,Z 686.003,A -85,B 0,C 180,E1 -28761.708,E2 -28761.708} C_VEL
LIN {X 0,Y 97.321,Z 678.207,A -85,B 0,C 180,E1 -28766.145,E2 -28766.145} C_VEL
LIN {X 0,Y 105.424,Z 668.518,A -85,B 0,C 180,E1 -28770.067,E2 -28770.067} C_VEL
LIN {X 0,Y 111.777,Z 659.446,A -85,B 0,C 180,E1 -28772.634,E2 -28772.634} C_VEL
LIN {X 0,Y 118.506,Z 647.872,A -85,B 0,C 180,E1 -28774.916,E2 -28774.916} C_VEL
LIN {X 0,Y 123.972,Z 635.87,A -85,B 0,C 180,E1 -28776.716,E2 -28776.716} C_VEL
LIN {X 0,Y 128.146,Z 623.742,A -85,B 0,C 180,E1 -28777.99,E2 -28777.99} C_VEL
LIN {X 0,Y 131.204,Z 610.569,A -85,B 0,C 180,E1 -28779.142,E2 -28779.142} C_VEL
LIN {X 0,Y 132.533,Z 601.062,A -85,B 0,C 180,E1 -28779.787,E2 -28779.787} C_VEL
LIN {X 0,Y 130.348,Z 595.018,A -85,B 0,C 180,E1 -28784.059,E2 -28784.059} C_VEL
LIN {X 0,Y 128.775,Z 591.38,A -85,B 0,C 180,E1 -28787.939,E2 -28787.939} C_VEL
LIN {X 0,Y 127.894,Z 588.897,A -85,B 0,C 180,E1 -28791.109,E2 -28791.109} C_VEL
LIN {X 0,Y 127.043,Z 585.942,A -85,B 0,C 180,E1 -28798.415,E2 -28798.415} C_VEL
LIN {X 0,Y 127.037,Z 586.476,A -85,B 0,C 180,E1 -28800.891,E2 -28800.891} C_VEL
LIN {X 0,Y 127.765,Z 588.861,A -85,B 0,C 180,E1 -28806.514,E2 -28806.514} C_VEL
LIN {X 0,Y 128.453,Z 592.526,A -85,B 0,C 180,E1 -28809.716,E2 -28809.716} C_VEL
LIN {X 0,Y 129.346,Z 597.188,A -85,B 0,C 180,E1 -28812.754,E2 -28812.754} C_VEL
LIN {X 0,Y 130.507,Z 603.502,A -85,B 0,C 180,E1 -28815.921,E2 -28815.921} C_VEL
LIN {X 0,Y 130.868,Z 605.554,A -85,B 0,C 180,E1 -28816.799,E2 -28816.799} C_VEL
LIN {X 0,Y 129.544,Z 620.932,A -85,B 0,C 180,E1 -28818.303,E2 -28818.303} C_VEL
LIN {X 0,Y 128.431,Z 627.088,A -85,B 0,C 180,E1 -28818.801,E2 -28818.801} C_VEL
LIN {X 0,Y 124.766,Z 639.807,A -85,B 0,C 180,E1 -28819.595,E2 -28819.595} C_VEL
LIN {X 0,Y 119.626,Z 652.759,A -85,B 0,C 180,E1 -28820.775,E2 -28820.775} C_VEL
LIN {X 0,Y 113.887,Z 664.025,A -85,B 0,C 180,E1 -28822.236,E2 -28822.236} C_VEL
LIN {X 0,Y 106.864,Z 674.959,A -85,B 0,C 180,E1 -28824.15,E2 -28824.15} C_VEL
LIN {X 0,Y 101.556,Z 682.109,A -85,B 0,C 180,E1 -28825.892,E2 -28825.892} C_VEL
LIN {X 0,Y 92.662,Z 692.169,A -85,B 0,C 180,E1 -28829.284,E2 -28829.284} C_VEL
LIN {X 0,Y 84.325,Z 700.328,A -85,B 0,C 180,E1 -28833.548,E2 -28833.548} C_VEL
LIN {X 0,Y 76.67,Z 706.926,A -85,B 0,C 180,E1 -28838.818,E2 -28838.818} C_VEL
LIN {X 0,Y 69.906,Z 712.225,A -85,B 0,C 180,E1 -28845.273,E2 -28845.273} C_VEL
LIN {X 0,Y 64.162,Z 716.379,A -85,B 0,C 180,E1 -28852.956,E2 -28852.956} C_VEL
LIN {X 0,Y 60.047,Z 719.544,A -85,B 0,C 180,E1 -28862.085,E2 -28862.085} C_VEL
LIN {X 0,Y 57.467,Z 722.281,A -85,B 0,C 180,E1 -28875.843,E2 -28875.843} C_VEL
LIN {X 0,Y 57.455,Z 723.063,A -85,B 0,C 180,E1 -28882.974,E2 -28882.974} C_VEL
LIN {X 0,Y 58.162,Z 723.428,A -85,B 0,C 180,E1 -28890,E2 -28890} C_VEL
LIN {X 0,Y 57.362,Z 722.624,A -85,B 0,C 180,E1 -28901.431,E2 -28901.431} C_VEL
LIN {X 0,Y 58.306,Z 721.064,A -85,B 0,C 180,E1 -28911.198,E2 -28911.198} C_VEL
LIN {X 0,Y 61.255,Z 718.508,A -85,B 0,C 180,E1 -28921.084,E2 -28921.084} C_VEL
LIN {X 0,Y 65.942,Z 714.991,A -85,B 0,C 180,E1 -28929.751,E2 -28929.751} C_VEL
LIN {X 0,Y 72.393,Z 710.15,A -85,B 0,C 180,E1 -28937.402,E2 -28937.402} C_VEL
LIN {X 0,Y 80.381,Z 703.621,A -85,B 0,C 180,E1 -28943.973,E2 -28943.973} C_VEL
LIN {X 0,Y 88.423,Z 696.235,A -85,B 0,C 180,E1 -28948.694,E2 -28948.694} C_VEL
LIN {X 0,Y 97.069,Z 687.141,A -85,B 0,C 180,E1 -28952.487,E2 -28952.487} C_VEL
LIN {X 0,Y 104.638,Z 677.849,A -85,B 0,C 180,E1 -28955.054,E2 -28955.054} C_VEL
LIN {X 0,Y 111.527,Z 667.498,A -85,B 0,C 180,E1 -28957.159,E2 -28957.159} C_VEL
LIN {X 0,Y 117.787,Z 656.054,A -85,B 0,C 180,E1 -28958.792,E2 -28958.792} C_VEL
LIN {X 0,Y 122.933,Z 644.192,A -85,B 0,C 180,E1 -28959.996,E2 -28959.996} C_VEL
LIN {X 0,Y 127.118,Z 631.126,A -85,B 0,C 180,E1 -28960.917,E2 -28960.917} C_VEL
LIN {X 0,Y 128.77,Z 624.031,A -85,B 0,C 180,E1 -28961.337,E2 -28961.337} C_VEL
LIN {X 0,Y 130.303,Z 610.338,A -85,B 0,C 180,E1 -28962.692,E2 -28962.692} C_VEL
LIN {X 0,Y 130.563,Z 604.945,A -85,B 0,C 180,E1 -28963.282,E2 -28963.282} C_VEL
LIN {X 0,Y 129.279,Z 598.014,A -85,B 0,C 180,E1 -28966.603,E2 -28966.603} C_VEL
LIN {X 0,Y 128.303,Z 592.974,A -85,B 0,C 180,E1 -28969.745,E2 -28969.745} C_VEL
LIN {X 0,Y 127.736,Z 590.033,A -85,B 0,C 180,E1 -28972.094,E2 -28972.094} C_VEL
LIN {X 0,Y 127.44,Z 588.379,A -85,B 0,C 180,E1 -28973.668,E2 -28973.668} C_VEL
LIN {X 0,Y 126.754,Z 585.616,A -85,B 0,C 180,E1 -28980,E2 -28980} C_VEL
LIN {X 0,Y 126.752,Z 585.62,A -85,B 0,C 180,E1 -28981.986,E2 -28981.986} C_VEL
LIN {X 0,Y 127.764,Z 589.161,A -85,B 0,C 180,E1 -28989.699,E2 -28989.699} C_VEL
LIN {X 0,Y 129.227,Z 592.926,A -85,B 0,C 180,E1 -28994.166,E2 -28994.166} C_VEL
LIN {X 0,Y 130.807,Z 596.736,A -85,B 0,C 180,E1 -28997.591,E2 -28997.591} C_VEL
LIN {X 0,Y 132.301,Z 601.042,A -85,B 0,C 180,E1 -29000.418,E2 -29000.418} C_VEL
LIN {X 0,Y 131.901,Z 604.364,A -85,B 0,C 180,E1 -29000.589,E2 -29000.589} C_VEL
LIN {X 0,Y 131.203,Z 608.234,A -85,B 0,C 180,E1 -29000.697,E2 -29000.697} C_VEL
LIN {X 0,Y 129.117,Z 615.844,A -85,B 0,C 180,E1 -29000.434,E2 -29000.434} C_VEL
LIN {X 0,Y 124.247,Z 628.761,A -85,B 0,C 180,E1 -28999.761,E2 -28999.761} C_VEL
LIN {X 0,Y 122.079,Z 634.207,A -85,B 0,C 180,E1 -29000.047,E2 -29000.047} C_VEL
LIN {X 0,Y 116.939,Z 645.907,A -85,B 0,C 180,E1 -29001.608,E2 -29001.608} C_VEL
LIN {X 0,Y 111.759,Z 655.189,A -85,B 0,C 180,E1 -29003.122,E2 -29003.122} C_VEL
LIN {X 0,Y 105.786,Z 664.221,A -85,B 0,C 180,E1 -29005.155,E2 -29005.155} C_VEL
LIN {X 0,Y 99.239,Z 672.616,A -85,B 0,C 180,E1 -29007.723,E2 -29007.723} C_VEL
LIN {X 0,Y 92.208,Z 680.329,A -85,B 0,C 180,E1 -29010.969,E2 -29010.969} C_VEL
LIN {X 0,Y 83.927,Z 687.981,A -85,B 0,C 180,E1 -29015.477,E2 -29015.477} C_VEL
LIN {X 0,Y 75.258,Z 694.774,A -85,B 0,C 180,E1 -29021.663,E2 -29021.663} C_VEL
LIN {X 0,Y 68.392,Z 699.374,A -85,B 0,C 180,E1 -29028.093,E2 -29028.093} C_VEL
LIN {X 0,Y 62.32,Z 702.908,A -85,B 0,C 180,E1 -29035.678,E2 -29035.678} C_VEL
LIN {X 0,Y 58.944,Z 704.727,A -85,B 0,C 180,E1 -29041.516,E2 -29041.516} C_VEL
LIN {X 0,Y 54.57,Z 706.997,A -85,B 0,C 180,E1 -29055.074,E2 -29055.074} C_VEL
LIN {X 0,Y 52.86,Z 707.818,A -85,B 0,C 180,E1 -29070,E2 -29070} C_VEL
LIN {X 0,Y 54.566,Z 707.038,A -85,B 0,C 180,E1 -29084.927,E2 -29084.927} C_VEL
LIN {X 0,Y 58.925,Z 704.812,A -85,B 0,C 180,E1 -29098.494,E2 -29098.494} C_VEL
LIN {X 0,Y 64.279,Z 701.97,A -85,B 0,C 180,E1 -29106.966,E2 -29106.966} C_VEL
LIN {X 0,Y 70.635,Z 698.131,A -85,B 0,C 180,E1 -29114.144,E2 -29114.144} C_VEL
LIN {X 0,Y 77.872,Z 693.037,A -85,B 0,C 180,E1 -29120.497,E2 -29120.497} C_VEL
LIN {X 0,Y 85.366,Z 686.989,A -85,B 0,C 180,E1 -29125.412,E2 -29125.412} C_VEL
LIN {X 0,Y 93.587,Z 679.193,A -85,B 0,C 180,E1 -29129.721,E2 -29129.721} C_VEL
LIN {X 0,Y 102.098,Z 669.504,A -85,B 0,C 180,E1 -29133.488,E2 -29133.488} C_VEL
LIN {X 0,Y 108.726,Z 660.431,A -85,B 0,C 180,E1 -29135.925,E2 -29135.925} C_VEL
LIN {X 0,Y 115.698,Z 648.857,A -85,B 0,C 180,E1 -29138.075,E2 -29138.075} C_VEL
LIN {X 0,Y 121.29,Z 637.033,A -85,B 0,C 180,E1 -29139.748,E2 -29139.748} C_VEL
LIN {X 0,Y 125.806,Z 624.292,A -85,B 0,C 180,E1 -29141.003,E2 -29141.003} C_VEL
LIN {X 0,Y 128.808,Z 611.801,A -85,B 0,C 180,E1 -29142.059,E2 -29142.059} C_VEL
LIN {X 0,Y 129.891,Z 604.955,A -85,B 0,C 180,E1 -29142.584,E2 -29142.584} C_VEL
LIN {X 0,Y 128.624,Z 600.926,A -85,B 0,C 180,E1 -29145.766,E2 -29145.766} C_VEL
LIN {X 0,Y 127.428,Z 597.776,A -85,B 0,C 180,E1 -29149.272,E2 -29149.272} C_VEL
LIN {X 0,Y 126.685,Z 595.517,A -85,B 0,C 180,E1 -29152.492,E2 -29152.492} C_VEL
LIN {X 0,Y 126.164,Z 593.108,A -85,B 0,C 180,E1 -29158.404,E2 -29158.404} C_VEL
LIN {X 0,Y 126.154,Z 593.505,A -85,B 0,C 180,E1 -29160.598,E2 -29160.598} C_VEL
LIN {X 0,Y 126.672,Z 595.616,A -85,B 0,C 180,E1 -29165.572,E2 -29165.572} C_VEL
LIN {X 0,Y 127.128,Z 598.833,A -85,B 0,C 180,E1 -29168.344,E2 -29168.344} C_VEL
LIN {X 0,Y 127.819,Z 603.379,A -85,B 0,C 180,E1 -29171.313,E2 -29171.313} C_VEL
LIN {X 0,Y 128.606,Z 608.854,A -85,B 0,C 180,E1 -29174.035,E2 -29174.035} C_VEL
LIN {X 0,Y 127.103,Z 621.928,A -85,B 0,C 180,E1 -29175.364,E2 -29175.364} C_VEL
LIN {X 0,Y 125.814,Z 628.019,A -85,B 0,C 180,E1 -29175.827,E2 -29175.827} C_VEL
LIN {X 0,Y 121.854,Z 640.792,A -85,B 0,C 180,E1 -29176.6,E2 -29176.6} C_VEL
LIN {X 0,Y 116.592,Z 653.281,A -85,B 0,C 180,E1 -29177.677,E2 -29177.677} C_VEL
LIN {X 0,Y 110.584,Z 664.343,A -85,B 0,C 180,E1 -29179.032,E2 -29179.032} C_VEL
LIN {X 0,Y 103.36,Z 675.042,A -85,B 0,C 180,E1 -29180.786,E2 -29180.786} C_VEL
LIN {X 0,Y 95.525,Z 684.722,A -85,B 0,C 180,E1 -29183.128,E2 -29183.128} C_VEL
LIN {X 0,Y 87.891,Z 692.679,A -85,B 0,C 180,E1 -29185.9,E2 -29185.9} C_VEL
LIN {X 0,Y 79.184,Z 700.509,A -85,B 0,C 180,E1 -29190.078,E2 -29190.078} C_VEL
LIN {X 0,Y 69.84,Z 707.806,A -85,B 0,C 180,E1 -29196.388,E2 -29196.388} C_VEL
LIN {X 0,Y 62.742,Z 712.713,A -85,B 0,C 180,E1 -29203.275,E2 -29203.275} C_VEL
LIN {X 0,Y 56.815,Z 716.52,A -85,B 0,C 180,E1 -29211.795,E2 -29211.795} C_VEL
LIN {X 0,Y 53.812,Z 718.536,A -85,B 0,C 180,E1 -29218.507,E2 -29218.507} C_VEL
LIN {X 0,Y 50.54,Z 721.273,A -85,B 0,C 180,E1 -29233.852,E2 -29233.852} C_VEL
LIN {X 0,Y 50.354,Z 722.056,A -85,B 0,C 180,E1 -29241.977,E2 -29241.977} C_VEL
LIN {X 0,Y 51.046,Z 722.428,A -85,B 0,C 180,E1 -29250,E2 -29250} C_VEL
LIN {X 0,Y 50.345,Z 721.693,A -85,B 0,C 180,E1 -29262.266,E2 -29262.266} C_VEL
LIN {X 0,Y 51.694,Z 720.056,A -85,B 0,C 180,E1 -29274.07,E2 -29274.07} C_VEL
LIN {X 0,Y 55.234,Z 717.498,A -85,B 0,C 180,E1 -29284.929,E2 -29284.929} C_VEL
LIN {X 0,Y 60.609,Z 713.983,A -85,B 0,C 180,E1 -29294.085,E2 -29294.085} C_VEL
LIN {X 0,Y 67.453,Z 709.354,A -85,B 0,C 180,E1 -29301.585,E2 -29301.585} C_VEL
LIN {X 0,Y 76.401,Z 702.615,A -85,B 0,C 180,E1 -29308.306,E2 -29308.306} C_VEL
LIN {X 0,Y 84.931,Z 695.229,A -85,B 0,C 180,E1 -29312.815,E2 -29312.815} C_VEL
LIN {X 0,Y 93.996,Z 686.139,A -85,B 0,C 180,E1 -29316.334,E2 -29316.334} C_VEL
LIN {X 0,Y 101.839,Z 676.845,A -85,B 0,C 180,E1 -29318.689,E2 -29318.689} C_VEL
LIN {X 0,Y 108.163,Z 667.784,A -85,B 0,C 180,E1 -29320.412,E2 -29320.412} C_VEL
LIN {X 0,Y 114.489,Z 656.84,A -85,B 0,C 180,E1 -29321.896,E2 -29321.896} C_VEL
LIN {X 0,Y 120.364,Z 643.982,A -85,B 0,C 180,E1 -29323.102,E2 -29323.102} C_VEL
LIN {X 0,Y 124.367,Z 632.352,A -85,B 0,C 180,E1 -29323.872,E2 -29323.872} C_VEL
LIN {X 0,Y 126.321,Z 624.539,A -85,B 0,C 180,E1 -29324.343,E2 -29324.343} C_VEL
LIN {X 0,Y 128.18,Z 610.639,A -85,B 0,C 180,E1 -29325.714,E2 -29325.714} C_VEL
LIN {X 0,Y 128.299,Z 608.387,A -85,B 0,C 180,E1 -29326.032,E2 -29326.032} C_VEL
LIN {X 0,Y 127.472,Z 602.816,A -85,B 0,C 180,E1 -29328.874,E2 -29328.874} C_VEL
LIN {X 0,Y 126.721,Z 597.543,A -85,B 0,C 180,E1 -29332.331,E2 -29332.331} C_VEL
LIN {X 0,Y 126.315,Z 595.042,A -85,B 0,C 180,E1 -29334.813,E2 -29334.813} C_VEL
LIN {X 0,Y 125.872,Z 592.796,A -85,B 0,C 180,E1 -29340,E2 -29340} C_VEL
LIN {X 0,Y 125.864,Z 592.854,A -85,B 0,C 180,E1 -29342,E2 -29342} C_VEL
LIN {X 0,Y 126.677,Z 596.038,A -85,B 0,C 180,E1 -29348.977,E2 -29348.977} C_VEL
LIN {X 0,Y 127.941,Z 599.65,A -85,B 0,C 180,E1 -29353.299,E2 -29353.299} C_VEL
LIN {X 0,Y 129.246,Z 603.533,A -85,B 0,C 180,E1 -29356.669,E2 -29356.669} C_VEL
LIN {X 0,Y 129.638,Z 605.076,A -85,B 0,C 180,E1 -29357.657,E2 -29357.657} C_VEL
LIN {X 0,Y 127.084,Z 618.187,A -85,B 0,C 180,E1 -29358.509,E2 -29358.509} C_VEL
LIN {X 0,Y 123.199,Z 631.221,A -85,B 0,C 180,E1 -29359.713,E2 -29359.713} C_VEL
LIN {X 0,Y 122.079,Z 634.207,A -85,B 0,C 180,E1 -29360.047,E2 -29360.047} C_VEL
LIN {X 0,Y 119.702,Z 639.6,A -85,B 0,C 180,E1 -29360.408,E2 -29360.408} C_VEL
LIN {X 0,Y 114.803,Z 648.179,A -85,B 0,C 180,E1 -29360.298,E2 -29360.298} C_VEL
LIN {X 0,Y 109.282,Z 656.393,A -85,B 0,C 180,E1 -29360.214,E2 -29360.214} C_VEL
LIN {X 0,Y 105.923,Z 661.143,A -85,B 0,C 180,E1 -29360.685,E2 -29360.685} C_VEL
LIN {X 0,Y 99.186,Z 670.089,A -85,B 0,C 180,E1 -29362.911,E2 -29362.911} C_VEL
LIN {X 0,Y 91.732,Z 678.416,A -85,B 0,C 180,E1 -29365.815,E2 -29365.815} C_VEL
LIN {X 0,Y 83.024,Z 686.511,A -85,B 0,C 180,E1 -29369.814,E2 -29369.814} C_VEL
LIN {X 0,Y 73.905,Z 693.607,A -85,B 0,C 180,E1 -29375.111,E2 -29375.111} C_VEL
LIN {X 0,Y 65.792,Z 698.964,A -85,B 0,C 180,E1 -29381.605,E2 -29381.605} C_VEL
LIN {X 0,Y 58.821,Z 702.844,A -85,B 0,C 180,E1 -29388.919,E2 -29388.919} C_VEL
LIN {X 0,Y 52.871,Z 705.716,A -85,B 0,C 180,E1 -29397.88,E2 -29397.88} C_VEL
LIN {X 0,Y 47.813,Z 707.986,A -85,B 0,C 180,E1 -29412.904,E2 -29412.904} C_VEL
LIN {X 0,Y 45.832,Z 708.806,A -85,B 0,C 180,E1 -29430,E2 -29430} C_VEL
LIN {X 0,Y 47.809,Z 708.026,A -85,B 0,C 180,E1 -29447.097,E2 -29447.097} C_VEL
LIN {X 0,Y 52.853,Z 705.799,A -85,B 0,C 180,E1 -29462.132,E2 -29462.132} C_VEL
LIN {X 0,Y 58.815,Z 702.957,A -85,B 0,C 180,E1 -29471.086,E2 -29471.086} C_VEL
LIN {X 0,Y 65.774,Z 699.118,A -85,B 0,C 180,E1 -29478.412,E2 -29478.412} C_VEL
LIN {X 0,Y 73.601,Z 694.023,A -85,B 0,C 180,E1 -29484.722,E2 -29484.722} C_VEL
LIN {X 0,Y 81.582,Z 687.975,A -85,B 0,C 180,E1 -29489.479,E2 -29489.479} C_VEL
LIN {X 0,Y 90.248,Z 680.179,A -85,B 0,C 180,E1 -29493.577,E2 -29493.577} C_VEL
LIN {X 0,Y 99.16,Z 670.489,A -85,B 0,C 180,E1 -29497.125,E2 -29497.125} C_VEL
LIN {X 0,Y 106.053,Z 661.415,A -85,B 0,C 180,E1 -29499.393,E2 -29499.393} C_VEL
LIN {X 0,Y 113.263,Z 649.841,A -85,B 0,C 180,E1 -29501.37,E2 -29501.37} C_VEL
LIN {X 0,Y 119.086,Z 637.909,A -85,B 0,C 180,E1 -29502.932,E2 -29502.932} C_VEL
LIN {X 0,Y 123.736,Z 625.136,A -85,B 0,C 180,E1 -29504.099,E2 -29504.099} C_VEL
LIN {X 0,Y 126.949,Z 612.184,A -85,B 0,C 180,E1 -29505.113,E2 -29505.113} C_VEL
LIN {X 0,Y 127.457,Z 609.162,A -85,B 0,C 180,E1 -29505.348,E2 -29505.348} C_VEL
LIN {X 0,Y 126.602,Z 605.767,A -85,B 0,C 180,E1 -29508.594,E2 -29508.594} C_VEL
LIN {X 0,Y 125.672,Z 602.393,A -85,B 0,C 180,E1 -29513.175,E2 -29513.175} C_VEL
LIN {X 0,Y 125.285,Z 600.268,A -85,B 0,C 180,E1 -29518.393,E2 -29518.393} C_VEL
LIN {X 0,Y 125.277,Z 600.754,A -85,B 0,C 180,E1 -29520.803,E2 -29520.803} C_VEL
LIN {X 0,Y 125.62,Z 602.494,A -85,B 0,C 180,E1 -29524.713,E2 -29524.713} C_VEL
LIN {X 0,Y 125.914,Z 605.511,A -85,B 0,C 180,E1 -29527.214,E2 -29527.214} C_VEL
LIN {X 0,Y 126.402,Z 610.555,A -85,B 0,C 180,E1 -29530.31,E2 -29530.31} C_VEL
LIN {X 0,Y 126.559,Z 612.31,A -85,B 0,C 180,E1 -29531.209,E2 -29531.209} C_VEL
LIN {X 0,Y 124.682,Z 624.375,A -85,B 0,C 180,E1 -29532.457,E2 -29532.457} C_VEL
LIN {X 0,Y 121.452,Z 635.822,A -85,B 0,C 180,E1 -29533.112,E2 -29533.112} C_VEL
LIN {X 0,Y 116.662,Z 647.941,A -85,B 0,C 180,E1 -29533.903,E2 -29533.903} C_VEL
LIN {X 0,Y 110.632,Z 659.727,A -85,B 0,C 180,E1 -29535.054,E2 -29535.054} C_VEL
LIN {X 0,Y 103.52,Z 670.756,A -85,B 0,C 180,E1 -29536.478,E2 -29536.478} C_VEL
LIN {X 0,Y 96.216,Z 680.122,A -85,B 0,C 180,E1 -29538.278,E2 -29538.278} C_VEL
LIN {X 0,Y 88.17,Z 688.661,A -85,B 0,C 180,E1 -29540.518,E2 -29540.518} C_VEL
LIN {X 0,Y 78.858,Z 697.061,A -85,B 0,C 180,E1 -29544.009,E2 -29544.009} C_VEL
LIN {X 0,Y 70.012,Z 703.887,A -85,B 0,C 180,E1 -29548.558,E2 -29548.558} C_VEL
LIN {X 0,Y 60.582,Z 710.215,A -85,B 0,C 180,E1 -29555.705,E2 -29555.705} C_VEL
LIN {X 0,Y 53.438,Z 714.368,A -85,B 0,C 180,E1 -29563.67,E2 -29563.67} C_VEL
LIN {X 0,Y 47.849,Z 717.529,A -85,B 0,C 180,E1 -29574.02,E2 -29574.02} C_VEL
LIN {X 0,Y 43.708,Z 720.266,A -85,B 0,C 180,E1 -29591.242,E2 -29591.242} C_VEL
LIN {X 0,Y 43.277,Z 721.049,A -85,B 0,C 180,E1 -29600.654,E2 -29600.654} C_VEL
LIN {X 0,Y 43.929,Z 721.427,A -85,B 0,C 180,E1 -29610,E2 -29610} C_VEL
LIN {X 0,Y 43.71,Z 720.235,A -85,B 0,C 180,E1 -29628.758,E2 -29628.758} C_VEL
LIN {X 0,Y 47.869,Z 717.468,A -85,B 0,C 180,E1 -29645.962,E2 -29645.962} C_VEL
LIN {X 0,Y 53.476,Z 714.284,A -85,B 0,C 180,E1 -29656.287,E2 -29656.287} C_VEL
LIN {X 0,Y 61.296,Z 709.605,A -85,B 0,C 180,E1 -29665.021,E2 -29665.021} C_VEL
LIN {X 0,Y 70.012,Z 703.714,A -85,B 0,C 180,E1 -29671.441,E2 -29671.441} C_VEL
LIN {X 0,Y 78.881,Z 696.855,A -85,B 0,C 180,E1 -29675.953,E2 -29675.953} C_VEL
LIN {X 0,Y 88.176,Z 688.404,A -85,B 0,C 180,E1 -29679.473,E2 -29679.473} C_VEL
LIN {X 0,Y 96.219,Z 679.792,A -85,B 0,C 180,E1 -29681.717,E2 -29681.717} C_VEL
LIN {X 0,Y 104.342,Z 669.157,A -85,B 0,C 180,E1 -29683.697,E2 -29683.697} C_VEL
LIN {X 0,Y 111.392,Z 657.847,A -85,B 0,C 180,E1 -29685.144,E2 -29685.144} C_VEL
LIN {X 0,Y 117.205,Z 646.043,A -85,B 0,C 180,E1 -29686.192,E2 -29686.192} C_VEL
LIN {X 0,Y 122.153,Z 632.679,A -85,B 0,C 180,E1 -29687.005,E2 -29687.005} C_VEL
LIN {X 0,Y 124.207,Z 625.216,A -85,B 0,C 180,E1 -29687.427,E2 -29687.427} C_VEL
LIN {X 0,Y 126.282,Z 612.048,A -85,B 0,C 180,E1 -29688.766,E2 -29688.766} C_VEL
LIN {X 0,Y 125.723,Z 606.026,A -85,B 0,C 180,E1 -29692.169,E2 -29692.169} C_VEL
LIN {X 0,Y 125.367,Z 602.603,A -85,B 0,C 180,E1 -29694.874,E2 -29694.874} C_VEL
LIN {X 0,Y 125.24,Z 601.723,A -85,B 0,C 180,E1 -29695.978,E2 -29695.978} C_VEL
LIN {X 0,Y 124.99,Z 599.978,A -85,B 0,C 180,E1 -29700,E2 -29700} C_VEL
LIN {X 0,Y 124.981,Z 600.05,A -85,B 0,C 180,E1 -29702.014,E2 -29702.014} C_VEL
LIN {X 0,Y 125.603,Z 602.91,A -85,B 0,C 180,E1 -29708.244,E2 -29708.244} C_VEL
LIN {X 0,Y 126.455,Z 606.01,A -85,B 0,C 180,E1 -29712.03,E2 -29712.03} C_VEL
LIN {X 0,Y 127.183,Z 608.896,A -85,B 0,C 180,E1 -29714.746,E2 -29714.746} C_VEL
LIN {X 0,Y 124.492,Z 621.239,A -85,B 0,C 180,E1 -29715.589,E2 -29715.589} C_VEL
LIN {X 0,Y 120.791,Z 632.839,A -85,B 0,C 180,E1 -29716.647,E2 -29716.647} C_VEL
LIN {X 0,Y 115.706,Z 644.563,A -85,B 0,C 180,E1 -29718.004,E2 -29718.004} C_VEL
LIN {X 0,Y 109.97,Z 654.911,A -85,B 0,C 180,E1 -29719.503,E2 -29719.503} C_VEL
LIN {X 0,Y 105.923,Z 661.143,A -85,B 0,C 180,E1 -29720.685,E2 -29720.685} C_VEL
LIN {X 0,Y 101.115,Z 667.287,A -85,B 0,C 180,E1 -29721.373,E2 -29721.373} C_VEL
LIN {X 0,Y 95.707,Z 673.089,A -85,B 0,C 180,E1 -29721.644,E2 -29721.644} C_VEL
LIN {X 0,Y 88.579,Z 679.84,A -85,B 0,C 180,E1 -29722.312,E2 -29722.312} C_VEL
LIN {X 0,Y 84.377,Z 683.595,A -85,B 0,C 180,E1 -29723.449,E2 -29723.449} C_VEL
LIN {X 0,Y 75.012,Z 691.157,A -85,B 0,C 180,E1 -29727.704,E2 -29727.704} C_VEL
LIN {X 0,Y 66.746,Z 696.753,A -85,B 0,C 180,E1 -29732.612,E2 -29732.612} C_VEL
LIN {X 0,Y 58.687,Z 701.352,A -85,B 0,C 180,E1 -29738.887,E2 -29738.887} C_VEL
LIN {X 0,Y 51.324,Z 704.887,A -85,B 0,C 180,E1 -29746.792,E2 -29746.792} C_VEL
LIN {X 0,Y 47.065,Z 706.705,A -85,B 0,C 180,E1 -29753.325,E2 -29753.325} C_VEL
LIN {X 0,Y 41.147,Z 708.974,A -85,B 0,C 180,E1 -29770.026,E2 -29770.026} C_VEL
LIN {X 0,Y 38.804,Z 709.794,A -85,B 0,C 180,E1 -29790,E2 -29790} C_VEL
LIN {X 0,Y 41.143,Z 709.014,A -85,B 0,C 180,E1 -29809.976,E2 -29809.976} C_VEL
LIN {X 0,Y 47.048,Z 706.787,A -85,B 0,C 180,E1 -29826.691,E2 -29826.691} C_VEL
LIN {X 0,Y 53.717,Z 703.944,A -85,B 0,C 180,E1 -29836.019,E2 -29836.019} C_VEL
LIN {X 0,Y 61.335,Z 700.105,A -85,B 0,C 180,E1 -29843.328,E2 -29843.328} C_VEL
LIN {X 0,Y 69.779,Z 695.01,A -85,B 0,C 180,E1 -29849.439,E2 -29849.439} C_VEL
LIN {X 0,Y 78.247,Z 688.961,A -85,B 0,C 180,E1 -29853.917,E2 -29853.917} C_VEL
LIN {X 0,Y 87.347,Z 681.165,A -85,B 0,C 180,E1 -29857.709,E2 -29857.709} C_VEL
LIN {X 0,Y 96.645,Z 671.474,A -85,B 0,C 180,E1 -29860.968,E2 -29860.968} C_VEL
LIN {X 0,Y 103.784,Z 662.402,A -85,B 0,C 180,E1 -29863.036,E2 -29863.036} C_VEL
LIN {X 0,Y 111.219,Z 650.822,A -85,B 0,C 180,E1 -29864.803,E2 -29864.803} C_VEL
LIN {X 0,Y 116.882,Z 639.628,A -85,B 0,C 180,E1 -29866.152,E2 -29866.152} C_VEL
LIN {X 0,Y 121.515,Z 627.645,A -85,B 0,C 180,E1 -29867.165,E2 -29867.165} C_VEL
LIN {X 0,Y 125.081,Z 614.294,A -85,B 0,C 180,E1 -29868.144,E2 -29868.144} C_VEL
LIN {X 0,Y 125.203,Z 613.53,A -85,B 0,C 180,E1 -29868.31,E2 -29868.31} C_VEL
LIN {X 0,Y 124.702,Z 610.703,A -85,B 0,C 180,E1 -29871.696,E2 -29871.696} C_VEL
LIN {X 0,Y 124.509,Z 609.219,A -85,B 0,C 180,E1 -29873.924,E2 -29873.924} C_VEL
LIN {X 0,Y 124.34,Z 607.437,A -85,B 0,C 180,E1 -29878.38,E2 -29878.38} C_VEL
LIN {X 0,Y 124.34,Z 607.908,A -85,B 0,C 180,E1 -29880.809,E2 -29880.809} C_VEL
LIN {X 0,Y 124.53,Z 609.221,A -85,B 0,C 180,E1 -29883.741,E2 -29883.741} C_VEL
LIN {X 0,Y 124.648,Z 613.253,A -85,B 0,C 180,E1 -29886.78,E2 -29886.78} C_VEL
LIN {X 0,Y 124.677,Z 615.946,A -85,B 0,C 180,E1 -29888.37,E2 -29888.37} C_VEL
LIN {X 0,Y 122.466,Z 626.893,A -85,B 0,C 180,E1 -29889.461,E2 -29889.461} C_VEL
LIN {X 0,Y 118.62,Z 638.674,A -85,B 0,C 180,E1 -29889.98,E2 -29889.98} C_VEL
LIN {X 0,Y 113.341,Z 650.749,A -85,B 0,C 180,E1 -29890.721,E2 -29890.721} C_VEL
LIN {X 0,Y 106.792,Z 662.349,A -85,B 0,C 180,E1 -29891.791,E2 -29891.791} C_VEL
LIN {X 0,Y 99.207,Z 673.048,A -85,B 0,C 180,E1 -29893.08,E2 -29893.08} C_VEL
LIN {X 0,Y 90.887,Z 682.729,A -85,B 0,C 180,E1 -29894.859,E2 -29894.859} C_VEL
LIN {X 0,Y 81.039,Z 692.074,A -85,B 0,C 180,E1 -29897.459,E2 -29897.459} C_VEL
LIN {X 0,Y 71.514,Z 699.652,A -85,B 0,C 180,E1 -29901,E2 -29901} C_VEL
LIN {X 0,Y 62.413,Z 705.793,A -85,B 0,C 180,E1 -29905.734,E2 -29905.734} C_VEL
LIN {X 0,Y 53.971,Z 710.71,A -85,B 0,C 180,E1 -29912.178,E2 -29912.178} C_VEL
LIN {X 0,Y 46.419,Z 714.509,A -85,B 0,C 180,E1 -29920.8,E2 -29920.8} C_VEL
LIN {X 0,Y 42.247,Z 716.52,A -85,B 0,C 180,E1 -29928.287,E2 -29928.287} C_VEL
LIN {X 0,Y 36.982,Z 719.257,A -85,B 0,C 180,E1 -29947.662,E2 -29947.662} C_VEL
LIN {X 0,Y 36.231,Z 720.043,A -85,B 0,C 180,E1 -29958.815,E2 -29958.815} C_VEL
LIN {X 0,Y 36.81,Z 720.426,A -85,B 0,C 180,E1 -29970,E2 -29970} C_VEL
LIN {X 0,Y 36.985,Z 719.225,A -85,B 0,C 180,E1 -29992.336,E2 -29992.336} C_VEL
LIN {X 0,Y 42.269,Z 716.458,A -85,B 0,C 180,E1 -30011.686,E2 -30011.686} C_VEL
LIN {X 0,Y 48.808,Z 713.278,A -85,B 0,C 180,E1 -30022.367,E2 -30022.367} C_VEL
LIN {X 0,Y 56.799,Z 709.003,A -85,B 0,C 180,E1 -30030.335,E2 -30030.335} C_VEL
LIN {X 0,Y 66.892,Z 702.708,A -85,B 0,C 180,E1 -30036.822,E2 -30036.822} C_VEL
LIN {X 0,Y 76.251,Z 695.849,A -85,B 0,C 180,E1 -30040.86,E2 -30040.86} C_VEL
LIN {X 0,Y 85.945,Z 687.404,A -85,B 0,C 180,E1 -30043.907,E2 -30043.907} C_VEL
LIN {X 0,Y 94.233,Z 678.79,A -85,B 0,C 180,E1 -30045.82,E2 -30045.82} C_VEL
LIN {X 0,Y 101.733,Z 669.338,A -85,B 0,C 180,E1 -30047.362,E2 -30047.362} C_VEL
LIN {X 0,Y 108.744,Z 658.62,A -85,B 0,C 180,E1 -30048.559,E2 -30048.559} C_VEL
LIN {X 0,Y 115.059,Z 646.517,A -85,B 0,C 180,E1 -30049.518,E2 -30049.518} C_VEL
LIN {X 0,Y 120.122,Z 633.604,A -85,B 0,C 180,E1 -30050.215,E2 -30050.215} C_VEL
LIN {X 0,Y 122.586,Z 625.159,A -85,B 0,C 180,E1 -30050.673,E2 -30050.673} C_VEL
LIN {X 0,Y 124.406,Z 615.526,A -85,B 0,C 180,E1 -30051.692,E2 -30051.692} C_VEL
LIN {X 0,Y 124.31,Z 611.042,A -85,B 0,C 180,E1 -30054.526,E2 -30054.526} C_VEL
LIN {X 0,Y 124.225,Z 608.65,A -85,B 0,C 180,E1 -30056.554,E2 -30056.554} C_VEL
LIN {X 0,Y 124.066,Z 607.128,A -85,B 0,C 180,E1 -30060,E2 -30060} C_VEL
LIN {X 0,Y 124.038,Z 607.227,A -85,B 0,C 180,E1 -30062.03,E2 -30062.03} C_VEL
LIN {X 0,Y 124.327,Z 609.58,A -85,B 0,C 180,E1 -30067.307,E2 -30067.307} C_VEL
LIN {X 0,Y 124.833,Z 612.596,A -85,B 0,C 180,E1 -30071.077,E2 -30071.077} C_VEL
LIN {X 0,Y 124.923,Z 613.493,A -85,B 0,C 180,E1 -30071.891,E2 -30071.891} C_VEL
LIN {X 0,Y 121.615,Z 626.163,A -85,B 0,C 180,E1 -30072.729,E2 -30072.729} C_VEL
LIN {X 0,Y 116.936,Z 638.775,A -85,B 0,C 180,E1 -30073.869,E2 -30073.869} C_VEL
LIN {X 0,Y 111.29,Z 650.128,A -85,B 0,C 180,E1 -30075.193,E2 -30075.193} C_VEL
LIN {X 0,Y 105.432,Z 659.593,A -85,B 0,C 180,E1 -30076.624,E2 -30076.624} C_VEL
LIN {X 0,Y 99.827,Z 667.244,A -85,B 0,C 180,E1 -30078.122,E2 -30078.122} C_VEL
LIN {X 0,Y 91.983,Z 676.254,A -85,B 0,C 180,E1 -30080.619,E2 -30080.619} C_VEL
LIN {X 0,Y 84.377,Z 683.595,A -85,B 0,C 180,E1 -30083.449,E2 -30083.449} C_VEL
LIN {X 0,Y 80.026,Z 687.174,A -85,B 0,C 180,E1 -30084.716,E2 -30084.716} C_VEL
LIN {X 0,Y 71.972,Z 692.714,A -85,B 0,C 180,E1 -30085.992,E2 -30085.992} C_VEL
LIN {X 0,Y 63.616,Z 697.618,A -85,B 0,C 180,E1 -30087.738,E2 -30087.738} C_VEL
LIN {X 0,Y 58.895,Z 700.148,A -85,B 0,C 180,E1 -30090.02,E2 -30090.02} C_VEL
LIN {X 0,Y 49.103,Z 704.822,A -85,B 0,C 180,E1 -30098.076,E2 -30098.076} C_VEL
LIN {X 0,Y 41.639,Z 707.694,A -85,B 0,C 180,E1 -30107.537,E2 -30107.537} C_VEL
LIN {X 0,Y 34.624,Z 709.963,A -85,B 0,C 180,E1 -30126.05,E2 -30126.05} C_VEL
LIN {X 0,Y 31.776,Z 710.782,A -85,B 0,C 180,E1 -30150,E2 -30150} C_VEL
LIN {X 0,Y 34.621,Z 710.002,A -85,B 0,C 180,E1 -30173.953,E2 -30173.953} C_VEL
LIN {X 0,Y 41.623,Z 707.775,A -85,B 0,C 180,E1 -30192.484,E2 -30192.484} C_VEL
LIN {X 0,Y 49.098,Z 704.931,A -85,B 0,C 180,E1 -30201.931,E2 -30201.931} C_VEL
LIN {X 0,Y 57.415,Z 701.092,A -85,B 0,C 180,E1 -30208.962,E2 -30208.962} C_VEL
LIN {X 0,Y 66.481,Z 695.997,A -85,B 0,C 180,E1 -30214.662,E2 -30214.662} C_VEL
LIN {X 0,Y 75.422,Z 689.948,A -85,B 0,C 180,E1 -30218.718,E2 -30218.718} C_VEL
LIN {X 0,Y 84.931,Z 682.151,A -85,B 0,C 180,E1 -30222.101,E2 -30222.101} C_VEL
LIN {X 0,Y 94.586,Z 672.46,A -85,B 0,C 180,E1 -30224.996,E2 -30224.996} C_VEL
LIN {X 0,Y 101.95,Z 663.389,A -85,B 0,C 180,E1 -30226.829,E2 -30226.829} C_VEL
LIN {X 0,Y 109.585,Z 651.807,A -85,B 0,C 180,E1 -30228.357,E2 -30228.357} C_VEL
LIN {X 0,Y 115.505,Z 640.392,A -85,B 0,C 180,E1 -30229.562,E2 -30229.562} C_VEL
LIN {X 0,Y 120.149,Z 628.625,A -85,B 0,C 180,E1 -30230.434,E2 -30230.434} C_VEL
LIN {X 0,Y 123.128,Z 618.324,A -85,B 0,C 180,E1 -30231.185,E2 -30231.185} C_VEL
LIN {X 0,Y 123.019,Z 615.964,A -85,B 0,C 180,E1 -30234.673,E2 -30234.673} C_VEL
LIN {X 0,Y 123.09,Z 614.551,A -85,B 0,C 180,E1 -30238.364,E2 -30238.364} C_VEL
LIN {X 0,Y 123.118,Z 615.144,A -85,B 0,C 180,E1 -30241.226,E2 -30241.226} C_VEL
LIN {X 0,Y 123.168,Z 616.024,A -85,B 0,C 180,E1 -30242.862,E2 -30242.862} C_VEL
LIN {X 0,Y 122.922,Z 619.669,A -85,B 0,C 180,E1 -30245.441,E2 -30245.441} C_VEL
LIN {X 0,Y 120.905,Z 628.003,A -85,B 0,C 180,E1 -30246.203,E2 -30246.203} C_VEL
LIN {X 0,Y 116.514,Z 640.44,A -85,B 0,C 180,E1 -30246.685,E2 -30246.685} C_VEL
LIN {X 0,Y 110.869,Z 652.332,A -85,B 0,C 180,E1 -30247.323,E2 -30247.323} C_VEL
LIN {X 0,Y 103.852,Z 663.958,A -85,B 0,C 180,E1 -30248.231,E2 -30248.231} C_VEL
LIN {X 0,Y 96.131,Z 674.174,A -85,B 0,C 180,E1 -30249.268,E2 -30249.268} C_VEL
LIN {X 0,Y 87.629,Z 683.419,A -85,B 0,C 180,E1 -30250.75,E2 -30250.75} C_VEL
LIN {X 0,Y 77.522,Z 692.454,A -85,B 0,C 180,E1 -30252.953,E2 -30252.953} C_VEL
LIN {X 0,Y 67.643,Z 699.79,A -85,B 0,C 180,E1 -30256.047,E2 -30256.047} C_VEL
LIN {X 0,Y 59.655,Z 704.789,A -85,B 0,C 180,E1 -30259.532,E2 -30259.532} C_VEL
LIN {X 0,Y 49.775,Z 710.091,A -85,B 0,C 180,E1 -30265.898,E2 -30265.898} C_VEL
LIN {X 0,Y 39.557,Z 714.545,A -85,B 0,C 180,E1 -30276.919,E2 -30276.919} C_VEL
LIN {X 0,Y 33.219,Z 717.074,A -85,B 0,C 180,E1 -30290.604,E2 -30290.604} C_VEL
LIN {X 0,Y 29.254,Z 719.038,A -85,B 0,C 180,E1 -30316.1,E2 -30316.1} C_VEL
LIN {X 0,Y 29.67,Z 719.422,A -85,B 0,C 180,E1 -30330,E2 -30330} C_VEL
LIN {X 0,Y 30.485,Z 718.218,A -85,B 0,C 180,E1 -30357.456,E2 -30357.456} C_VEL
LIN {X 0,Y 37.224,Z 715.449,A -85,B 0,C 180,E1 -30379.043,E2 -30379.043} C_VEL
LIN {X 0,Y 44.804,Z 712.272,A -85,B 0,C 180,E1 -30389.623,E2 -30389.623} C_VEL
LIN {X 0,Y 53.488,Z 708.069,A -85,B 0,C 180,E1 -30396.887,E2 -30396.887} C_VEL
LIN {X 0,Y 64.413,Z 701.7,A -85,B 0,C 180,E1 -30402.685,E2 -30402.685} C_VEL
LIN {X 0,Y 74.211,Z 694.84,A -85,B 0,C 180,E1 -30406.091,E2 -30406.091} C_VEL
LIN {X 0,Y 84.252,Z 686.402,A -85,B 0,C 180,E1 -30408.557,E2 -30408.557} C_VEL
LIN {X 0,Y 92.744,Z 677.784,A -85,B 0,C 180,E1 -30410.095,E2 -30410.095} C_VEL
LIN {X 0,Y 100.42,Z 668.337,A -85,B 0,C 180,E1 -30411.314,E2 -30411.314} C_VEL
LIN {X 0,Y 108.122,Z 656.654,A -85,B 0,C 180,E1 -30412.377,E2 -30412.377} C_VEL
LIN {X 0,Y 113.905,Z 645.662,A -85,B 0,C 180,E1 -30413.035,E2 -30413.035} C_VEL
LIN {X 0,Y 118.803,Z 633.546,A -85,B 0,C 180,E1 -30413.561,E2 -30413.561} C_VEL
LIN {X 0,Y 121.389,Z 624.975,A -85,B 0,C 180,E1 -30413.999,E2 -30413.999} C_VEL
LIN {X 0,Y 122.656,Z 619.315,A -85,B 0,C 180,E1 -30414.623,E2 -30414.623} C_VEL
LIN {X 0,Y 122.899,Z 615.342,A -85,B 0,C 180,E1 -30417.542,E2 -30417.542} C_VEL
LIN {X 0,Y 122.842,Z 614.301,A -85,B 0,C 180,E1 -30420,E2 -30420} C_VEL
LIN {X 0,Y 122.786,Z 614.371,A -85,B 0,C 180,E1 -30422.05,E2 -30422.05} C_VEL
LIN {X 0,Y 122.763,Z 616.519,A -85,B 0,C 180,E1 -30426.802,E2 -30426.802} C_VEL
LIN {X 0,Y 122.86,Z 617.983,A -85,B 0,C 180,E1 -30428.849,E2 -30428.849} C_VEL
LIN {X 0,Y 119.311,Z 630.078,A -85,B 0,C 180,E1 -30429.703,E2 -30429.703} C_VEL
LIN {X 0,Y 114.421,Z 641.959,A -85,B 0,C 180,E1 -30430.664,E2 -30430.664} C_VEL
LIN {X 0,Y 109.026,Z 652.183,A -85,B 0,C 180,E1 -30431.754,E2 -30431.754} C_VEL
LIN {X 0,Y 101.977,Z 662.901,A -85,B 0,C 180,E1 -30433.235,E2 -30433.235} C_VEL
LIN {X 0,Y 94.604,Z 672.071,A -85,B 0,C 180,E1 -30435.044,E2 -30435.044} C_VEL
LIN {X 0,Y 86.54,Z 680.397,A -85,B 0,C 180,E1 -30437.408,E2 -30437.408} C_VEL
LIN {X 0,Y 77.008,Z 688.492,A -85,B 0,C 180,E1 -30440.702,E2 -30440.702} C_VEL
LIN {X 0,Y 66.818,Z 695.587,A -85,B 0,C 180,E1 -30445.202,E2 -30445.202} C_VEL
LIN {X 0,Y 58.895,Z 700.148,A -85,B 0,C 180,E1 -30450.02,E2 -30450.02} C_VEL
LIN {X 0,Y 54.142,Z 702.48,A -85,B 0,C 180,E1 -30452.668,E2 -30452.668} C_VEL
LIN {X 0,Y 45.384,Z 705.934,A -85,B 0,C 180,E1 -30456.284,E2 -30456.284} C_VEL
LIN {X 0,Y 36.715,Z 708.737,A -85,B 0,C 180,E1 -30461.777,E2 -30461.777} C_VEL
LIN {X 0,Y 32.437,Z 709.907,A -85,B 0,C 180,E1 -30468.161,E2 -30468.161} C_VEL
LIN {X 0,Y 28.345,Z 710.952,A -85,B 0,C 180,E1 -30480.273,E2 -30480.273} C_VEL
LIN {X 0,Y 24.748,Z 711.771,A -85,B 0,C 180,E1 -30510,E2 -30510} C_VEL
LIN {X 0,Y 28.342,Z 710.99,A -85,B 0,C 180,E1 -30539.731,E2 -30539.731} C_VEL
LIN {X 0,Y 36.746,Z 708.763,A -85,B 0,C 180,E1 -30559.908,E2 -30559.908} C_VEL
LIN {X 0,Y 45.105,Z 705.919,A -85,B 0,C 180,E1 -30568.977,E2 -30568.977} C_VEL
LIN {X 0,Y 54.127,Z 702.079,A -85,B 0,C 180,E1 -30575.35,E2 -30575.35} C_VEL
LIN {X 0,Y 63.79,Z 696.983,A -85,B 0,C 180,E1 -30580.376,E2 -30580.376} C_VEL
LIN {X 0,Y 73.164,Z 690.934,A -85,B 0,C 180,E1 -30583.853,E2 -30583.853} C_VEL
LIN {X 0,Y 83.04,Z 683.136,A -85,B 0,C 180,E1 -30586.72,E2 -30586.72} C_VEL
LIN {X 0,Y 93.015,Z 673.445,A -85,B 0,C 180,E1 -30589.182,E2 -30589.182} C_VEL
LIN {X 0,Y 100.579,Z 664.376,A -85,B 0,C 180,E1 -30590.74,E2 -30590.74} C_VEL
LIN {X 0,Y 108.385,Z 652.791,A -85,B 0,C 180,E1 -30591.992,E2 -30591.992} C_VEL
LIN {X 0,Y 114.582,Z 641.073,A -85,B 0,C 180,E1 -30593.046,E2 -30593.046} C_VEL
LIN {X 0,Y 119.342,Z 629.123,A -85,B 0,C 180,E1 -30593.801,E2 -30593.801} C_VEL
LIN {X 0,Y 121.14,Z 623.334,A -85,B 0,C 180,E1 -30594.256,E2 -30594.256} C_VEL
LIN {X 0,Y 121.435,Z 621.575,A -85,B 0,C 180,E1 -30598.342,E2 -30598.342} C_VEL
LIN {X 0,Y 121.479,Z 622.009,A -85,B 0,C 180,E1 -30600.829,E2 -30600.829} C_VEL
LIN {X 0,Y 121.405,Z 622.736,A -85,B 0,C 180,E1 -30601.808,E2 -30601.808} C_VEL
LIN {X 0,Y 121.272,Z 623.563,A -85,B 0,C 180,E1 -30602.454,E2 -30602.454} C_VEL
LIN {X 0,Y 119.625,Z 629.304,A -85,B 0,C 180,E1 -30602.884,E2 -30602.884} C_VEL
LIN {X 0,Y 114.895,Z 641.751,A -85,B 0,C 180,E1 -30603.269,E2 -30603.269} C_VEL
LIN {X 0,Y 108.544,Z 654.317,A -85,B 0,C 180,E1 -30603.788,E2 -30603.788} C_VEL
LIN {X 0,Y 101.335,Z 665.406,A -85,B 0,C 180,E1 -30604.485,E2 -30604.485} C_VEL
LIN {X 0,Y 93.509,Z 675.15,A -85,B 0,C 180,E1 -30605.238,E2 -30605.238} C_VEL
LIN {X 0,Y 84.856,Z 684.072,A -85,B 0,C 180,E1 -30606.36,E2 -30606.36} C_VEL
LIN {X 0,Y 74.527,Z 692.792,A -85,B 0,C 180,E1 -30608.052,E2 -30608.052} C_VEL
LIN {X 0,Y 64.34,Z 699.837,A -85,B 0,C 180,E1 -30610.56,E2 -30610.56} C_VEL
LIN {X 0,Y 54.369,Z 705.543,A -85,B 0,C 180,E1 -30614.194,E2 -30614.194} C_VEL
LIN {X 0,Y 44.739,Z 710.072,A -85,B 0,C 180,E1 -30619.523,E2 -30619.523} C_VEL
LIN {X 0,Y 35.713,Z 713.538,A -85,B 0,C 180,E1 -30627.683,E2 -30627.683} C_VEL
LIN {X 0,Y 28.047,Z 716.066,A -85,B 0,C 180,E1 -30641.261,E2 -30641.261} C_VEL
LIN {X 0,Y 22.393,Z 718.035,A -85,B 0,C 180,E1 -30671.709,E2 -30671.709} C_VEL
LIN {X 0,Y 22.518,Z 718.417,A -85,B 0,C 180,E1 -30690,E2 -30690} C_VEL
